(* CODESYS project tc3_vision.library
   TcLibraryId: Beckhoff Automation GmbH|Tc3_Vision|4.0.7.4
   Company: Beckhoff Automation GmbH
   DefaultNamespace: Tc3_Vision
   Version: 4.0.7.4
   Placeholder: Tc3_Vision
   Title: Tc3_Vision

Project tree, tasks and I/O mapping:
  Version/
    global variables Global_Version
  Function Blocks/
    Image Acquisition/
      function block FB_VN_GevCameraControl [ST]: ClearImageQueue, CloseCamera, FB_exit, FB_init, GetCalibPatternRef, GetCameraMatrix, GetCurrentImage, GetCurrentImageUndistorted, GetCurrentImageWithGvspInfo, GetCurrentImageWithGvspInfoUndistorted, GetCurrentImageWithTimestamps, GetDistortionCoefficients, GetLastImageFromQueue, GetOmittedImagesNum, GetRotationMatrix, GetState, GetTranslationVector, InitializeCamera, OpenCamera, Reset, ResetCameraFeatures, SetCameraMatrix, SetDistortionCoefficients, SetRotationMatrix, SetTranslationVector, StartAcquisition, StopAcquisition, TriggerImage
      function block FB_VN_FileSourceControl [ST]: FB_exit, FB_init, GetCurrentImage, GetCurrentImageAndFileName, StartAcquisition, StopAcquisition, Reset, GetState, TriggerImage, TriggerImageExp, TriggerImageByName
      function block FB_VN_SimpleCameraControl [ST]: FB_exit, FB_init, GetCurrentImage, GetState, Reset, StartAcquisition, StopAcquisition, TriggerImage
    File Access/
      function block FB_VN_InitializeFunction [ST]: FB_exit, FB_init
      function block FB_VN_ReadCalibrationPattern [ST]: FB_exit, FB_init
      function block FB_VN_ReadCalibrationResult [ST]: FB_exit, FB_init
      function block FB_VN_ReadContainer [ST]: FB_exit, FB_init
      function block FB_VN_ReadNeuralNetwork [ST]: FB_exit, FB_init
      function block FB_VN_ReadImage [ST]: FB_exit, FB_init
      function block FB_VN_ReadMlModel [ST]: FB_exit, FB_init
      function block FB_VN_WriteCalibrationResult [ST]: FB_exit, FB_init
      function block FB_VN_WriteContainer [ST]: FB_exit, FB_init
      function block FB_VN_WriteImage [ST]: FB_exit, FB_init
      function block FB_VN_WriteMlModel [ST]: FB_exit, FB_init
    Camera Register Access/
      function block FB_VN_ReadRegister_UDINT [ST]: FB_exit, FB_init
      function block FB_VN_WriteRegister_UDINT [ST]: FB_exit, FB_init
      function block FB_VN_ReadRegister_ULINT [ST]: FB_exit, FB_init
      function block FB_VN_WriteRegister_ULINT [ST]: FB_exit, FB_init
      function block FB_VN_ReadMemory [ST]: FB_exit, FB_init
      function block FB_VN_WriteMemory [ST]: FB_exit, FB_init
      function block FB_VN_ReadRegister_REAL [ST]: FB_exit, FB_init
      function block FB_VN_WriteRegister_REAL [ST]: FB_exit, FB_init
    Image Processing/
      function block FB_VN_GeneralizedHoughBallard [ST]: FB_exit, FB_init, Detect, SetCannyThreshold, SetInvAccuRatio, SetLevels, SetMinDist, SetTemplate, SetVotesThreshold
      function block FB_VN_SSIM [ST]: FB_exit, FB_init, Compute, SetReference
  Functions/
    Control Functions/
      function F_VN_StartAbsWatchdog [ST]
      function F_VN_StartAbsWatchdogExp [ST]
      function F_VN_StartRelWatchdog [ST]
      function F_VN_StartRelWatchdogExp [ST]
      function F_VN_StopWatchdog [ST]
    Image Segmentation/
      function F_VN_AdaptiveThreshold [ST]
      function F_VN_AdaptiveThresholdExp [ST]
      function F_VN_CheckColorRange [ST]
      function F_VN_DoubleThreshold [ST]
      function F_VN_SauvolaThreshold [ST]
      function F_VN_Threshold [ST]
      function F_VN_WatershedSegmentationExp [ST]
    Algebraic Container Operations/
      function F_VN_AddContainers [ST]
      F_VN_AddToContainerElements/
        function F_VN_AddToContainerElements_DINT [ST]
        function F_VN_AddToContainerElements_INT [ST]
        function F_VN_AddToContainerElements_LREAL [ST]
        function F_VN_AddToContainerElements_REAL [ST]
        function F_VN_AddToContainerElements_SINT [ST]
        function F_VN_AddToContainerElements_TcVnKeyPoint [ST]
        function F_VN_AddToContainerElements_TcVnPoint2_DINT [ST]
        function F_VN_AddToContainerElements_TcVnPoint2_LREAL [ST]
        function F_VN_AddToContainerElements_TcVnPoint2_REAL [ST]
        function F_VN_AddToContainerElements_TcVnPoint3_LREAL [ST]
        function F_VN_AddToContainerElements_TcVnPoint3_REAL [ST]
        function F_VN_AddToContainerElements_TcVnRectangle_DINT [ST]
        function F_VN_AddToContainerElements_TcVnRotatedRectangle [ST]
        function F_VN_AddToContainerElements_TcVnVector2_DINT [ST]
        function F_VN_AddToContainerElements_TcVnVector2_INT [ST]
        function F_VN_AddToContainerElements_TcVnVector2_REAL [ST]
        function F_VN_AddToContainerElements_TcVnVector2_SINT [ST]
        function F_VN_AddToContainerElements_TcVnVector2_UINT [ST]
        function F_VN_AddToContainerElements_TcVnVector2_USINT [ST]
        function F_VN_AddToContainerElements_TcVnVector3_INT [ST]
        function F_VN_AddToContainerElements_TcVnVector3_REAL [ST]
        function F_VN_AddToContainerElements_TcVnVector3_SINT [ST]
        function F_VN_AddToContainerElements_TcVnVector3_UINT [ST]
        function F_VN_AddToContainerElements_TcVnVector3_USINT [ST]
        function F_VN_AddToContainerElements_TcVnVector4_DINT [ST]
        function F_VN_AddToContainerElements_TcVnVector4_INT [ST]
        function F_VN_AddToContainerElements_TcVnVector4_LREAL [ST]
        function F_VN_AddToContainerElements_TcVnVector4_REAL [ST]
        function F_VN_AddToContainerElements_TcVnVector4_SINT [ST]
        function F_VN_AddToContainerElements_TcVnVector4_UINT [ST]
        function F_VN_AddToContainerElements_TcVnVector4_USINT [ST]
        function F_VN_AddToContainerElements_UDINT [ST]
        function F_VN_AddToContainerElements_UINT [ST]
        function F_VN_AddToContainerElements_ULINT [ST]
        function F_VN_AddToContainerElements_USINT [ST]
      function F_VN_BitwiseAndContainers [ST]
      function F_VN_BitwiseNotContainer [ST]
      function F_VN_BitwiseOrContainers [ST]
      function F_VN_BitwiseXorContainers [ST]
      function F_VN_DivideContainers [ST]
      function F_VN_DivideContainersExp [ST]
      function F_VN_MaxContainer [ST]
      function F_VN_MinContainer [ST]
      function F_VN_MultiplyContainers [ST]
      function F_VN_MultiplyWithContainerElements1 [ST]
      function F_VN_MultiplyWithContainerElements2 [ST]
      function F_VN_MultiplyWithContainerElements3 [ST]
      function F_VN_MultiplyWithContainerElements4 [ST]
      function F_VN_NegateContainer [ST]
      function F_VN_SubtractContainers [ST]
    Algebraic Image Operations/
      function F_VN_AddImages [ST]
      function F_VN_AddImagesWeighted [ST]
      function F_VN_AddImagesWeightedExp [ST]
      function F_VN_AddScalarToImage [ST]
      function F_VN_AddVectorToImage [ST]
      function F_VN_BitwiseAndImages [ST]
      function F_VN_BitwiseAndImagesExp [ST]
      function F_VN_BitwiseAndScalarWithImage [ST]
      function F_VN_BitwiseAndVectorWithImage [ST]
      function F_VN_BitwiseNotImage [ST]
      function F_VN_BitwiseNotImageExp [ST]
      function F_VN_BitwiseOrImages [ST]
      function F_VN_BitwiseOrImagesExp [ST]
      function F_VN_BitwiseOrScalarWithImage [ST]
      function F_VN_BitwiseOrVectorWithImage [ST]
      function F_VN_BitwiseXorImages [ST]
      function F_VN_BitwiseXorImagesExp [ST]
      function F_VN_BitwiseXorScalarWithImage [ST]
      function F_VN_BitwiseXorVectorWithImage [ST]
      function F_VN_BlendImages [ST]
      function F_VN_DivideImageByScalar [ST]
      function F_VN_DivideImageByVector [ST]
      function F_VN_DivideImages [ST]
      function F_VN_DivideScalarByImage [ST]
      function F_VN_DivideVectorByImage [ST]
      function F_VN_ElementwiseExp [ST]
      function F_VN_ElementwiseLog [ST]
      function F_VN_MaxImage [ST]
      function F_VN_MaxImageExp [ST]
      function F_VN_MaxImageWithScalar [ST]
      function F_VN_MaxImageWithScalarExp [ST]
      function F_VN_MaxImageWithVector [ST]
      function F_VN_MaxImageWithVectorExp [ST]
      function F_VN_MinImage [ST]
      function F_VN_MinImageExp [ST]
      function F_VN_MinImageWithScalar [ST]
      function F_VN_MinImageWithScalarExp [ST]
      function F_VN_MinImageWithVector [ST]
      function F_VN_MinImageWithVectorExp [ST]
      function F_VN_MultiplyImages [ST]
      function F_VN_MultiplyImageWithScalar [ST]
      function F_VN_MultiplyImageWithVector [ST]
      function F_VN_SubtractImageFromScalar [ST]
      function F_VN_SubtractImageFromVector [ST]
      function F_VN_SubtractImages [ST]
      function F_VN_SubtractScalarFromImage [ST]
      function F_VN_SubtractVectorFromImage [ST]
    Image Analysis/
      Object Detection/
        function F_VN_AdjustActiveContour [ST]
        function F_VN_DetectBlobs [ST]
        function F_VN_DetectBlobsExp [ST]
        function F_VN_FindContourHierarchyExp [ST]
        function F_VN_FindContours [ST]
        function F_VN_FindContoursExp [ST]
        function F_VN_HoughCircles [ST]
        function F_VN_HoughCirclesExp [ST]
        function F_VN_HoughLines [ST]
        function F_VN_HoughLinesExp [ST]
        function F_VN_HoughLinesP [ST]
        function F_VN_HoughLinesPExp [ST]
        function F_VN_MatchImageHuMoments [ST]
        function F_VN_MatchTemplate [ST]
        function F_VN_MatchTemplateExp [ST]
        function F_VN_MatchTemplateAndEvaluate [ST]
        function F_VN_MatchTemplateAndEvaluateExp [ST]
      function F_VN_CannyEdgeDetection [ST]
      function F_VN_CannyEdgeDetectionExp [ST]
      function F_VN_ConnectedComponents [ST]
      function F_VN_ConnectedComponentsExp [ST]
      function F_VN_ConnectedComponentsWithStats [ST]
      function F_VN_ConnectedComponentsWithStatsExp [ST]
      function F_VN_CountNonZeroPixels [ST]
      function F_VN_DistanceTransformation [ST]
      function F_VN_DistanceTransformationExp [ST]
      function F_VN_GetConnectedComponent [ST]
      function F_VN_GetConnectedComponentExp [ST]
      function F_VN_ImageAbsoluteAverage [ST]
      function F_VN_ImageAverage [ST]
      function F_VN_ImageAverageExp [ST]
      function F_VN_ImageAverageStdDev [ST]
      function F_VN_ImageAverageStdDevExp [ST]
      function F_VN_ImageCenterOfMass [ST]
      function F_VN_ImageCenterOfMassExp [ST]
      function F_VN_ImageMedian [ST]
      function F_VN_ImageMedianExp [ST]
      function F_VN_ImageMoments [ST]
      function F_VN_MaxPixelValue [ST]
      function F_VN_MaxPixelValueExp [ST]
      function F_VN_MinPixelValue [ST]
      function F_VN_MinPixelValueExp [ST]
      function F_VN_RegionOrientation [ST]
      function F_VN_RegionOrientationExp [ST]
      function F_VN_UprightInnerRectangle [ST]
      function F_VN_UprightInnerRectangleExp [ST]
    Measurement/
      function F_VN_AdjustSearchWindowOrientationToLinearEdge [ST]
      function F_VN_ClosestPointsBF [ST]
      function F_VN_LocateCircularArc [ST]
      function F_VN_LocateCircularArcExp [ST]
      function F_VN_LocateEdge [ST]
      function F_VN_LocateEdgeExp [ST]
      function F_VN_LocateEdges [ST]
      function F_VN_LocateEdgesExp [ST]
      function F_VN_LocateEllipse [ST]
      function F_VN_LocateEllipseExp [ST]
      function F_VN_MeasureAngleBetweenEdges [ST]
      function F_VN_MeasureAngleBetweenEdgesExp [ST]
      function F_VN_MeasureEdgeDistance [ST]
      function F_VN_MeasureEdgeDistanceExp [ST]
      function F_VN_MeasureMinEdgeDistance [ST]
      function F_VN_MeasureMinEdgeDistanceExp [ST]
    Basic Container Operations/
      function F_VN_AdvanceIterator [ST]
      F_VN_AppendToContainer/
        function F_VN_AppendToContainer_ITcVnContainer [ST]
        function F_VN_AppendToContainer_ITcVnForwardIterator [ST]
        function F_VN_AppendToContainer_DINT [ST]
        function F_VN_AppendToContainer_INT [ST]
        function F_VN_AppendToContainer_ITcVnImage [ST]
        function F_VN_AppendToContainer_LREAL [ST]
        function F_VN_AppendToContainer_REAL [ST]
        function F_VN_AppendToContainer_SINT [ST]
        function F_VN_AppendToContainer_TcVnDMatch [ST]
        function F_VN_AppendToContainer_TcVnKeyPoint [ST]
        function F_VN_AppendToContainer_TcVnPoint2_DINT [ST]
        function F_VN_AppendToContainer_TcVnPoint2_LREAL [ST]
        function F_VN_AppendToContainer_TcVnPoint2_REAL [ST]
        function F_VN_AppendToContainer_TcVnPoint3_LREAL [ST]
        function F_VN_AppendToContainer_TcVnPoint3_REAL [ST]
        function F_VN_AppendToContainer_TcVnRectangle_DINT [ST]
        function F_VN_AppendToContainer_TcVnRotatedRectangle [ST]
        function F_VN_AppendToContainer_TcVnVector2_DINT [ST]
        function F_VN_AppendToContainer_TcVnVector2_INT [ST]
        function F_VN_AppendToContainer_TcVnVector2_REAL [ST]
        function F_VN_AppendToContainer_TcVnVector2_SINT [ST]
        function F_VN_AppendToContainer_TcVnVector2_UINT [ST]
        function F_VN_AppendToContainer_TcVnVector2_USINT [ST]
        function F_VN_AppendToContainer_TcVnVector3_INT [ST]
        function F_VN_AppendToContainer_TcVnVector3_REAL [ST]
        function F_VN_AppendToContainer_TcVnVector3_SINT [ST]
        function F_VN_AppendToContainer_TcVnVector3_UINT [ST]
        function F_VN_AppendToContainer_TcVnVector3_USINT [ST]
        function F_VN_AppendToContainer_TcVnVector4_DINT [ST]
        function F_VN_AppendToContainer_TcVnVector4_INT [ST]
        function F_VN_AppendToContainer_TcVnVector4_LREAL [ST]
        function F_VN_AppendToContainer_TcVnVector4_REAL [ST]
        function F_VN_AppendToContainer_TcVnVector4_SINT [ST]
        function F_VN_AppendToContainer_TcVnVector4_UINT [ST]
        function F_VN_AppendToContainer_TcVnVector4_USINT [ST]
        function F_VN_AppendToContainer_UDINT [ST]
        function F_VN_AppendToContainer_UINT [ST]
        function F_VN_AppendToContainer_ULINT [ST]
        function F_VN_AppendToContainer_USINT [ST]
      function F_VN_CheckIfEmpty [ST]
      function F_VN_CheckIfIteratorIsAtEnd [ST]
      function F_VN_ConvertContainerType [ST]
      function F_VN_CopyContainer [ST]
      function F_VN_CopyContainerElementsConditional_ITcVnContainer [ST]
      function F_VN_CopyContainerElementsConditional_ITcVnForwardIterator [ST]
      function F_VN_CreateContainer [ST]
      function F_VN_CreateContainerFromArray [ST]
      function F_VN_EraseFromContainer [ST]
      function F_VN_ExportContainer [ST]
      function F_VN_ExportContainer_String [ST]
      function F_VN_ExportContainerSize [ST]
      function F_VN_ExportSubContainer [ST]
      function F_VN_ExportSubContainer_String [ST]
      function F_VN_ExportSubContainerSize [ST]
      function F_VN_ExtractContainerRange [ST]
      F_VN_FillContainer/
        function F_VN_FillContainer_DINT [ST]
        function F_VN_FillContainer_INT [ST]
        function F_VN_FillContainer_ITcVnImage [ST]
        function F_VN_FillContainer_LREAL [ST]
        function F_VN_FillContainer_REAL [ST]
        function F_VN_FillContainer_SINT [ST]
        function F_VN_FillContainer_TcVnDMatch [ST]
        function F_VN_FillContainer_TcVnKeyPoint [ST]
        function F_VN_FillContainer_TcVnPoint2_DINT [ST]
        function F_VN_FillContainer_TcVnPoint2_LREAL [ST]
        function F_VN_FillContainer_TcVnPoint2_REAL [ST]
        function F_VN_FillContainer_TcVnPoint3_LREAL [ST]
        function F_VN_FillContainer_TcVnPoint3_REAL [ST]
        function F_VN_FillContainer_TcVnRectangle_DINT [ST]
        function F_VN_FillContainer_TcVnRotatedRectangle [ST]
        function F_VN_FillContainer_TcVnVector2_DINT [ST]
        function F_VN_FillContainer_TcVnVector2_INT [ST]
        function F_VN_FillContainer_TcVnVector2_REAL [ST]
        function F_VN_FillContainer_TcVnVector2_SINT [ST]
        function F_VN_FillContainer_TcVnVector2_UINT [ST]
        function F_VN_FillContainer_TcVnVector2_USINT [ST]
        function F_VN_FillContainer_TcVnVector3_INT [ST]
        function F_VN_FillContainer_TcVnVector3_REAL [ST]
        function F_VN_FillContainer_TcVnVector3_SINT [ST]
        function F_VN_FillContainer_TcVnVector3_UINT [ST]
        function F_VN_FillContainer_TcVnVector3_USINT [ST]
        function F_VN_FillContainer_TcVnVector4_DINT [ST]
        function F_VN_FillContainer_TcVnVector4_INT [ST]
        function F_VN_FillContainer_TcVnVector4_LREAL [ST]
        function F_VN_FillContainer_TcVnVector4_REAL [ST]
        function F_VN_FillContainer_TcVnVector4_SINT [ST]
        function F_VN_FillContainer_TcVnVector4_UINT [ST]
        function F_VN_FillContainer_TcVnVector4_USINT [ST]
        function F_VN_FillContainer_UDINT [ST]
        function F_VN_FillContainer_UINT [ST]
        function F_VN_FillContainer_ULINT [ST]
        function F_VN_FillContainer_USINT [ST]
      F_VN_FillContainerExp/
        function F_VN_FillContainerExp_DINT [ST]
        function F_VN_FillContainerExp_INT [ST]
        function F_VN_FillContainerExp_ITcVnImage [ST]
        function F_VN_FillContainerExp_LREAL [ST]
        function F_VN_FillContainerExp_REAL [ST]
        function F_VN_FillContainerExp_SINT [ST]
        function F_VN_FillContainerExp_TcVnDMatch [ST]
        function F_VN_FillContainerExp_TcVnKeyPoint [ST]
        function F_VN_FillContainerExp_TcVnPoint2_DINT [ST]
        function F_VN_FillContainerExp_TcVnPoint2_LREAL [ST]
        function F_VN_FillContainerExp_TcVnPoint2_REAL [ST]
        function F_VN_FillContainerExp_TcVnPoint3_LREAL [ST]
        function F_VN_FillContainerExp_TcVnPoint3_REAL [ST]
        function F_VN_FillContainerExp_TcVnRectangle_DINT [ST]
        function F_VN_FillContainerExp_TcVnRotatedRectangle [ST]
        function F_VN_FillContainerExp_TcVnVector2_DINT [ST]
        function F_VN_FillContainerExp_TcVnVector2_INT [ST]
        function F_VN_FillContainerExp_TcVnVector2_REAL [ST]
        function F_VN_FillContainerExp_TcVnVector2_SINT [ST]
        function F_VN_FillContainerExp_TcVnVector2_UINT [ST]
        function F_VN_FillContainerExp_TcVnVector2_USINT [ST]
        function F_VN_FillContainerExp_TcVnVector3_INT [ST]
        function F_VN_FillContainerExp_TcVnVector3_REAL [ST]
        function F_VN_FillContainerExp_TcVnVector3_SINT [ST]
        function F_VN_FillContainerExp_TcVnVector3_UINT [ST]
        function F_VN_FillContainerExp_TcVnVector3_USINT [ST]
        function F_VN_FillContainerExp_TcVnVector4_DINT [ST]
        function F_VN_FillContainerExp_TcVnVector4_INT [ST]
        function F_VN_FillContainerExp_TcVnVector4_LREAL [ST]
        function F_VN_FillContainerExp_TcVnVector4_REAL [ST]
        function F_VN_FillContainerExp_TcVnVector4_SINT [ST]
        function F_VN_FillContainerExp_TcVnVector4_UINT [ST]
        function F_VN_FillContainerExp_TcVnVector4_USINT [ST]
        function F_VN_FillContainerExp_UDINT [ST]
        function F_VN_FillContainerExp_UINT [ST]
        function F_VN_FillContainerExp_ULINT [ST]
        function F_VN_FillContainerExp_USINT [ST]
      F_VN_GetAt/
        function F_VN_GetAt_ITcVnContainer [ST]
        function F_VN_GetAt_DINT [ST]
        function F_VN_GetAt_INT [ST]
        function F_VN_GetAt_ITcVnImage [ST]
        function F_VN_GetAt_LREAL [ST]
        function F_VN_GetAt_REAL [ST]
        function F_VN_GetAt_SINT [ST]
        function F_VN_GetAt_TcVnDMatch [ST]
        function F_VN_GetAt_TcVnKeyPoint [ST]
        function F_VN_GetAt_TcVnPoint2_DINT [ST]
        function F_VN_GetAt_TcVnPoint2_LREAL [ST]
        function F_VN_GetAt_TcVnPoint2_REAL [ST]
        function F_VN_GetAt_TcVnPoint3_LREAL [ST]
        function F_VN_GetAt_TcVnPoint3_REAL [ST]
        function F_VN_GetAt_TcVnRectangle_DINT [ST]
        function F_VN_GetAt_TcVnRotatedRectangle [ST]
        function F_VN_GetAt_TcVnVector2_DINT [ST]
        function F_VN_GetAt_TcVnVector2_INT [ST]
        function F_VN_GetAt_TcVnVector2_REAL [ST]
        function F_VN_GetAt_TcVnVector2_SINT [ST]
        function F_VN_GetAt_TcVnVector2_UINT [ST]
        function F_VN_GetAt_TcVnVector2_USINT [ST]
        function F_VN_GetAt_TcVnVector3_INT [ST]
        function F_VN_GetAt_TcVnVector3_REAL [ST]
        function F_VN_GetAt_TcVnVector3_SINT [ST]
        function F_VN_GetAt_TcVnVector3_UINT [ST]
        function F_VN_GetAt_TcVnVector3_USINT [ST]
        function F_VN_GetAt_TcVnVector4_DINT [ST]
        function F_VN_GetAt_TcVnVector4_INT [ST]
        function F_VN_GetAt_TcVnVector4_LREAL [ST]
        function F_VN_GetAt_TcVnVector4_REAL [ST]
        function F_VN_GetAt_TcVnVector4_SINT [ST]
        function F_VN_GetAt_TcVnVector4_UINT [ST]
        function F_VN_GetAt_TcVnVector4_USINT [ST]
        function F_VN_GetAt_UDINT [ST]
        function F_VN_GetAt_UINT [ST]
        function F_VN_GetAt_ULINT [ST]
        function F_VN_GetAt_USINT [ST]
      function F_VN_GetContainer [ST]
      function F_VN_GetContainerExp [ST]
      function F_VN_GetForwardIterator [ST]
      function F_VN_GetNumberOfElements [ST]
      function F_VN_GetRandomAccessIterator [ST]
      function F_VN_IncrementIterator [ST]
      F_VN_InsertIntoContainer/
        function F_VN_InsertIntoContainer_ITcVnContainer [ST]
        function F_VN_InsertIntoContainer_ITcVnForwardIterator [ST]
        function F_VN_InsertIntoContainer_DINT [ST]
        function F_VN_InsertIntoContainer_INT [ST]
        function F_VN_InsertIntoContainer_ITcVnImage [ST]
        function F_VN_InsertIntoContainer_LREAL [ST]
        function F_VN_InsertIntoContainer_REAL [ST]
        function F_VN_InsertIntoContainer_SINT [ST]
        function F_VN_InsertIntoContainer_TcVnDMatch [ST]
        function F_VN_InsertIntoContainer_TcVnKeyPoint [ST]
        function F_VN_InsertIntoContainer_TcVnPoint2_DINT [ST]
        function F_VN_InsertIntoContainer_TcVnPoint2_LREAL [ST]
        function F_VN_InsertIntoContainer_TcVnPoint2_REAL [ST]
        function F_VN_InsertIntoContainer_TcVnPoint3_LREAL [ST]
        function F_VN_InsertIntoContainer_TcVnPoint3_REAL [ST]
        function F_VN_InsertIntoContainer_TcVnRectangle_DINT [ST]
        function F_VN_InsertIntoContainer_TcVnRotatedRectangle [ST]
        function F_VN_InsertIntoContainer_TcVnVector2_DINT [ST]
        function F_VN_InsertIntoContainer_TcVnVector2_INT [ST]
        function F_VN_InsertIntoContainer_TcVnVector2_REAL [ST]
        function F_VN_InsertIntoContainer_TcVnVector2_SINT [ST]
        function F_VN_InsertIntoContainer_TcVnVector2_UINT [ST]
        function F_VN_InsertIntoContainer_TcVnVector2_USINT [ST]
        function F_VN_InsertIntoContainer_TcVnVector3_INT [ST]
        function F_VN_InsertIntoContainer_TcVnVector3_REAL [ST]
        function F_VN_InsertIntoContainer_TcVnVector3_SINT [ST]
        function F_VN_InsertIntoContainer_TcVnVector3_UINT [ST]
        function F_VN_InsertIntoContainer_TcVnVector3_USINT [ST]
        function F_VN_InsertIntoContainer_TcVnVector4_DINT [ST]
        function F_VN_InsertIntoContainer_TcVnVector4_INT [ST]
        function F_VN_InsertIntoContainer_TcVnVector4_LREAL [ST]
        function F_VN_InsertIntoContainer_TcVnVector4_REAL [ST]
        function F_VN_InsertIntoContainer_TcVnVector4_SINT [ST]
        function F_VN_InsertIntoContainer_TcVnVector4_UINT [ST]
        function F_VN_InsertIntoContainer_TcVnVector4_USINT [ST]
        function F_VN_InsertIntoContainer_UDINT [ST]
        function F_VN_InsertIntoContainer_UINT [ST]
        function F_VN_InsertIntoContainer_ULINT [ST]
        function F_VN_InsertIntoContainer_USINT [ST]
      function F_VN_IteratorDistance [ST]
      function F_VN_ReserveContainerMemory [ST]
      function F_VN_ReverseContainer [ST]
      F_VN_SetAt/
        function F_VN_SetAt_ITcVnContainer [ST]
        function F_VN_SetAt_DINT [ST]
        function F_VN_SetAt_INT [ST]
        function F_VN_SetAt_ITcVnImage [ST]
        function F_VN_SetAt_LREAL [ST]
        function F_VN_SetAt_REAL [ST]
        function F_VN_SetAt_SINT [ST]
        function F_VN_SetAt_TcVnDMatch [ST]
        function F_VN_SetAt_TcVnKeyPoint [ST]
        function F_VN_SetAt_TcVnPoint2_DINT [ST]
        function F_VN_SetAt_TcVnPoint2_LREAL [ST]
        function F_VN_SetAt_TcVnPoint2_REAL [ST]
        function F_VN_SetAt_TcVnPoint3_LREAL [ST]
        function F_VN_SetAt_TcVnPoint3_REAL [ST]
        function F_VN_SetAt_TcVnRectangle_DINT [ST]
        function F_VN_SetAt_TcVnRotatedRectangle [ST]
        function F_VN_SetAt_TcVnVector2_DINT [ST]
        function F_VN_SetAt_TcVnVector2_INT [ST]
        function F_VN_SetAt_TcVnVector2_REAL [ST]
        function F_VN_SetAt_TcVnVector2_SINT [ST]
        function F_VN_SetAt_TcVnVector2_UINT [ST]
        function F_VN_SetAt_TcVnVector2_USINT [ST]
        function F_VN_SetAt_TcVnVector3_INT [ST]
        function F_VN_SetAt_TcVnVector3_REAL [ST]
        function F_VN_SetAt_TcVnVector3_SINT [ST]
        function F_VN_SetAt_TcVnVector3_UINT [ST]
        function F_VN_SetAt_TcVnVector3_USINT [ST]
        function F_VN_SetAt_TcVnVector4_DINT [ST]
        function F_VN_SetAt_TcVnVector4_INT [ST]
        function F_VN_SetAt_TcVnVector4_LREAL [ST]
        function F_VN_SetAt_TcVnVector4_REAL [ST]
        function F_VN_SetAt_TcVnVector4_SINT [ST]
        function F_VN_SetAt_TcVnVector4_UINT [ST]
        function F_VN_SetAt_TcVnVector4_USINT [ST]
        function F_VN_SetAt_UDINT [ST]
        function F_VN_SetAt_UINT [ST]
        function F_VN_SetAt_ULINT [ST]
        function F_VN_SetAt_USINT [ST]
      function F_VN_SetContainer [ST]
      function F_VN_SetIteratorToBegin [ST]
    Geometric and Coordinate Transformations/
      function F_VN_AlignRotatedImageRegion [ST]
      function F_VN_AlignRotatedImageRegionExp [ST]
      function F_VN_ApplyRotationToAffineTransformation [ST]
      function F_VN_ApplyRotationToAffineTransformationExp [ST]
      function F_VN_ApplyScalingToAffineTransformation [ST]
      function F_VN_ApplyScalingToAffineTransformationExp [ST]
      function F_VN_ApplyTranslationToAffineTransformation [ST]
      function F_VN_ApplyTranslationToAffineTransformationExp [ST]
      function F_VN_ApplyYAxisInversionToAffineTransformation [ST]
      function F_VN_ApplyYAxisInversionToAffineTransformationExp [ST]
      Calibration/
        function F_VN_CalibrateCamera [ST]
        function F_VN_CalibrateCameraExp [ST]
        function F_VN_CalibrateCameraExp2 [ST]
        function F_VN_CalibrateCameraExp3 [ST]
        function F_VN_CalibrateCameraManually [ST]
        function F_VN_CalibrateCameraManuallyExp [ST]
        function F_VN_CalibrateCameraPlanar [ST]
        function F_VN_CalibrateCameraPlanarExp [ST]
        function F_VN_CalibrateLinescanCamera [ST]
        function F_VN_CalibrateLinescanCameraExp [ST]
        function F_VN_CompensateLensDistortion [ST]
        function F_VN_CompensateLensDistortionExp1 [ST]
        function F_VN_CompensateLensDistortionExp2 [ST]
        function F_VN_CompensateLensDistortionForPoints [ST]
        function F_VN_CompensateLensDistortionForPointsExp1 [ST]
        function F_VN_CompensateLensDistortionForPointsExp2 [ST]
        function F_VN_DetectPatternPoints [ST]
        function F_VN_DetectPatternPointsExp [ST]
        function F_VN_GenerateCalibrationPatternReferencePoints [ST]
        function F_VN_ImagePointsWorldDistance [ST]
        function F_VN_SolvePnP [ST]
        function F_VN_SolvePnPExp [ST]
        function F_VN_SortDetectedPatternPoints [ST]
        function F_VN_TransformCoordinatesPlanar_Container [ST]
        function F_VN_TransformCoordinatesPlanar_Point [ST]
        function F_VN_TransformCoordinatesImageToWorld_Container [ST]
        function F_VN_TransformCoordinatesImageToWorld_Point [ST]
        function F_VN_TransformCoordinatesWorldToImage_Container [ST]
        function F_VN_TransformCoordinatesWorldToImage_Point [ST]
      function F_VN_ConvertCartesianToPolarAngleImage [ST]
      function F_VN_ConvertCartesianToPolarAngleImageExp [ST]
      function F_VN_ConvertCartesianToPolarAngles [ST]
      function F_VN_ConvertCartesianToPolarAnglesExp [ST]
      function F_VN_ConvertCartesianToPolarImages [ST]
      function F_VN_ConvertCartesianToPolarImagesExp [ST]
      function F_VN_ConvertCartesianToPolarMagnitudeImage [ST]
      function F_VN_ConvertCartesianToPolarMagnitudes [ST]
      function F_VN_ConvertCartesianToPolarPoints [ST]
      function F_VN_ConvertCartesianToPolarPointsExp [ST]
      function F_VN_ConvertPolarToCartesianImages [ST]
      function F_VN_ConvertPolarToCartesianImagesExp [ST]
      function F_VN_ConvertPolarToCartesianPoints [ST]
      function F_VN_ConvertPolarToCartesianPointsExp [ST]
      function F_VN_DecomposeAffineTransformation [ST]
      function F_VN_DecomposeAffineTransformationExp [ST]
      function F_VN_DecomposeHomography [ST]
      function F_VN_DecomposeHomographyExp [ST]
      function F_VN_FlipImage [ST]
      function F_VN_GenerateAffineTransformationUnitMatrix2D [ST]
      function F_VN_GetAffineTransformation [ST]
      function F_VN_GetAffineTransformation2D [ST]
      function F_VN_GetAffineTransformation2DExp [ST]
      function F_VN_GetPerspectiveTransformation [ST]
      function F_VN_Homography [ST]
      function F_VN_HomographyExp [ST]
      function F_VN_InvertAffineTransformation [ST]
      function F_VN_PerspectiveTransformation [ST]
      function F_VN_PyramidDown [ST]
      function F_VN_PyramidUp [ST]
      function F_VN_RemapImageToLogPolarSpace [ST]
      function F_VN_RemapImageToLogPolarSpaceExp [ST]
      function F_VN_RemapImageToLogPolarSpaceExp2 [ST]
      function F_VN_RemapImageToPolarSpace [ST]
      function F_VN_RemapImageToPolarSpaceExp [ST]
      function F_VN_RemapImageToPolarSpaceExp2 [ST]
      function F_VN_ResizeImage [ST]
      function F_VN_ResizeImageExp [ST]
      function F_VN_RotateImage [ST]
      function F_VN_RotateImageExp [ST]
      function F_VN_RotateImageExp2 [ST]
      function F_VN_WarpAffine [ST]
      function F_VN_WarpAffineExp [ST]
      function F_VN_WarpAffine_Container [ST]
      function F_VN_WarpAffine_Point [ST]
      function F_VN_WarpAffine_Rectangle [ST]
      function F_VN_WarpPerspective [ST]
      function F_VN_WarpPerspective_Container [ST]
      function F_VN_WarpPerspectiveExp [ST]
      function F_VN_WarpPerspective_Point [ST]
      function F_VN_WarpPerspective_Rectangle [ST]
    Image Color and Contrast Processing/
      function F_VN_ApplyColorMap [ST]
      function F_VN_ApplyLut [ST]
      function F_VN_Clahe [ST]
      function F_VN_ClaheExp [ST]
      function F_VN_ConvertColorSpace [ST]
      function F_VN_GenerateColorMap [ST]
      function F_VN_GenerateCustomColorMap [ST]
      function F_VN_Histogram [ST]
      function F_VN_HistogramExp [ST]
      function F_VN_HistogramEqualization [ST]
      function F_VN_HistogramEqualizationExp [ST]
      function F_VN_InvertImageColor [ST]
      function F_VN_InvertImageColorExp [ST]
      function F_VN_NormalizeImage [ST]
      function F_VN_NormalizeImageExp [ST]
      function F_VN_NormalizeImageForDisplay [ST]
      function F_VN_ReferenceColorSimilarity_ITcVnColorModel [ST]
      function F_VN_ReferenceColorSimilarityExp_ITcVnColorModel [ST]
      function F_VN_ReferenceColorSimilarity_ITcVnMlModel [ST]
      function F_VN_ReferenceColorSimilarityExp_ITcVnMlModel [ST]
      function F_VN_ReferenceColorSimilarity_TcVnVector3_LREAL [ST]
      function F_VN_ReferenceColorSimilarityExp_TcVnVector3_LREAL [ST]
      function F_VN_TrainImageColor [ST]
      function F_VN_TrainImageColorExp [ST]
      function F_VN_TrainImageColorExp2 [ST]
      function F_VN_TrainImageColor_ITcVnMlModel [ST]
      function F_VN_TrainImageColorExp_ITcVnMlModel [ST]
      function F_VN_TrainImageColorExp2_ITcVnMlModel [ST]
      function F_VN_WhiteBalance [ST]
    Contour Analysis/
      function F_VN_ApproximatePolygon [ST]
      function F_VN_CheckIfPointIsInsideContour [ST]
      function F_VN_ContourArea [ST]
      function F_VN_ContourCenterOfMass [ST]
      function F_VN_ContourCircularity [ST]
      function F_VN_ContourCircularityExp [ST]
      function F_VN_ContourConvexity [ST]
      function F_VN_ContourEccentricity [ST]
      function F_VN_ContourElongation [ST]
      function F_VN_ContourExtremePoint [ST]
      function F_VN_ContourInertiaRatio [ST]
      function F_VN_ContourMoments [ST]
      function F_VN_ContourOrientation [ST]
      function F_VN_ContourOrientationExp [ST]
      function F_VN_ContourPerimeter [ST]
      function F_VN_ContourRoundness [ST]
      function F_VN_ConvexHullPoints [ST]
      function F_VN_ConvexHullPointsExp [ST]
      function F_VN_ConvexityDefects [ST]
      function F_VN_CustomElementWiseContainerOperation_ITcVnContainer [ST]
      function F_VN_CustomElementWiseContainerOperation_ITcVnForwardIterator [ST]
      function F_VN_EnclosingCircle [ST]
      function F_VN_EnclosingRectangle [ST]
      function F_VN_EnclosingTriangle [ST]
      function F_VN_FitEllipse [ST]
      function F_VN_FitLine [ST]
      function F_VN_FitLineExp [ST]
      function F_VN_FourierDescriptors [ST]
      function F_VN_MatchContours [ST]
      function F_VN_MatchContoursExp [ST]
      function F_VN_MatchContours1vsN [ST]
      function F_VN_MatchContours1vsNExp [ST]
      function F_VN_UprightBoundingRectangle [ST]
    Image Filtering/
      function F_VN_BilateralFilter [ST]
      function F_VN_BilateralFilterExp [ST]
      function F_VN_BoxFilter [ST]
      function F_VN_BoxFilterExp [ST]
      function F_VN_BrightBorderObjects [ST]
      function F_VN_CreateStructuringElement [ST]
      function F_VN_CustomFilter [ST]
      function F_VN_CustomFilterExp [ST]
      function F_VN_DarkBorderObjects [ST]
      function F_VN_FillHoles [ST]
      function F_VN_GaussianFilter [ST]
      function F_VN_GaussianFilterExp [ST]
      function F_VN_LaplacianFilter [ST]
      function F_VN_LaplacianFilterExp [ST]
      function F_VN_LocalMaxima [ST]
      function F_VN_LocalMinima [ST]
      function F_VN_MedianFilter [ST]
      function F_VN_MorphologicalOperator [ST]
      function F_VN_RemoveLocalMaxima [ST]
      function F_VN_RemoveLocalMinima [ST]
      function F_VN_ScharrFilter [ST]
      function F_VN_ScharrFilterExp [ST]
      function F_VN_SeparableCustomFilter [ST]
      function F_VN_SeparableCustomFilterExp [ST]
      function F_VN_SobelFilter [ST]
      function F_VN_SobelFilterExp [ST]
      function F_VN_VarianceFilter [ST]
      function F_VN_VarianceFilterExp [ST]
    Miscellaneous/
      function F_VN_CheckFunctionInitialization [ST]
      function F_VN_ClipLineToBoundary [ST]
      function F_VN_ClipLineToBoundary_ITcVnImage [ST]
      function F_VN_ClipLineToBoundary_TcVnRectangle_DINT [ST]
      function F_VN_ConvertITcUnknownToITcVnBitmapExport [ST]
      function F_VN_ConvertITcUnknownToITcVnContainer [ST]
      function F_VN_ConvertITcUnknownToITcVnImage [ST]
      function F_VN_ConvertITcUnknownToITcVnMlModel [ST]
      function F_VN_DeinitializeFunction [ST]
      function F_VN_GetTimestamp [ST]
      function F_VN_HuMomentInvariants [ST]
      function F_VN_InitMatrixStruct [ST]
      function F_VN_InvertMatrix3x3 [ST]
      function F_VN_LineIntersectionPoint [ST]
      function F_VN_LineIntersectionPointAndAngle [ST]
      function F_VN_MultiplyMatrices [ST]
      function F_VN_OrthogonalVector_TcVnVector2_DINT [ST]
      function F_VN_OrthogonalVector_TcVnVector2_LREAL [ST]
      function F_VN_OrthogonalVector_TcVnVector2_REAL [ST]
      function F_VN_PointToLineDistance_TcVnPoint2_DINT [ST]
      function F_VN_PointToLineDistance_TcVnPoint2_LREAL [ST]
      function F_VN_PointToLineDistance_TcVnPoint2_REAL [ST]
      function F_VN_PointToPointDirection_TcVnPoint2_DINT [ST]
      function F_VN_PointToPointDirection_TcVnPoint2_LREAL [ST]
      function F_VN_PointToPointDirection_TcVnPoint2_REAL [ST]
      function F_VN_PointToPointDistance_TcVnPoint2_DINT [ST]
      function F_VN_PointToPointDistance_TcVnPoint2_LREAL [ST]
      function F_VN_PointToPointDistance_TcVnPoint2_REAL [ST]
      function F_VN_RotatedRectangleCorners [ST]
      function F_VN_RotatedRectangleIntersection [ST]
      function F_VN_SetRngSeed [ST]
      function F_VN_UpdateTimestamp [ST]
    Basic Image Operations/
      function F_VN_CombineImageChannels [ST]
      function F_VN_ConvertElementType [ST]
      function F_VN_ConvertElementTypeExp [ST]
      function F_VN_CopyImage [ST]
      function F_VN_CopyImageRegion [ST]
      function F_VN_CopyImageRegionToRegion [ST]
      function F_VN_CopyIntoDisplayableImage [ST]
      function F_VN_CreateAssociatedImage [ST]
      function F_VN_CreateEmptyImage [ST]
      function F_VN_CreateImage [ST]
      function F_VN_CreateNDimensionalImage [ST]
      function F_VN_CreateImageAndSetPixels [ST]
      function F_VN_CreateNDimensionalImageAndSetPixels [ST]
      function F_VN_CreateImageFromArray [ST]
      function F_VN_CreateNDimensionalImageFromArray [ST]
      function F_VN_ExportImage [ST]
      function F_VN_ExportImageSize [ST]
      function F_VN_ExportImageAsBmp [ST]
      function F_VN_ExportImageAsBmpExp [ST]
      function F_VN_ExportImageAsBmpSize [ST]
      function F_VN_ExportImageAsBmpSizeExp [ST]
      function F_VN_FuseImages [ST]
      function F_VN_FuseImagesArray [ST]
      function F_VN_GetImageChannel [ST]
      function F_VN_GetImageHeight [ST]
      function F_VN_GetImageInfo [ST]
      function F_VN_GetImageWidth [ST]
      function F_VN_GetLayoutInfo [ST]
      function F_VN_GetPixel [ST]
      function F_VN_GetPixelFormat [ST]
      function F_VN_GetRoi [ST]
      function F_VN_MixImageChannels [ST]
      function F_VN_PadImageBorder [ST]
      function F_VN_PadImageBorderExp [ST]
      function F_VN_ReinterpretUnsupportedImage [ST]
      function F_VN_ResetRoi [ST]
      function F_VN_SetImageChannel [ST]
      function F_VN_SetPixel [ST]
      function F_VN_SetPixels [ST]
      function F_VN_SetPixelsExp [ST]
      function F_VN_SetRoi [ST]
      function F_VN_SetRoi_TcVnRectangle_DINT [ST]
      function F_VN_SetRoi_TcVnRectangle_UDINT [ST]
      function F_VN_SplitImageChannels [ST]
      function F_VN_TransformIntoDisplayableImage [ST]
      function F_VN_TransformIntoDisplayableImageExp [ST]
    Container Statistics/
      function F_VN_ContainerAverage [ST]
      function F_VN_ContainerAverageElementwise2 [ST]
      function F_VN_ContainerAverageElementwise3 [ST]
      function F_VN_ContainerAverageElementwise4 [ST]
      function F_VN_ContainerAverageVariance [ST]
      function F_VN_ContainerAverageVarianceElementwise2 [ST]
      function F_VN_ContainerAverageVarianceElementwise3 [ST]
      function F_VN_ContainerAverageVarianceElementwise4 [ST]
      function F_VN_MaxElement [ST]
      F_VN_MaxElementElementwise/
        function F_VN_MaxElementElementwise_DINT [ST]
        function F_VN_MaxElementElementwise_INT [ST]
        function F_VN_MaxElementElementwise_LREAL [ST]
        function F_VN_MaxElementElementwise_REAL [ST]
        function F_VN_MaxElementElementwise_SINT [ST]
        function F_VN_MaxElementElementwise_TcVnPoint2_DINT [ST]
        function F_VN_MaxElementElementwise_TcVnPoint2_LREAL [ST]
        function F_VN_MaxElementElementwise_TcVnPoint2_REAL [ST]
        function F_VN_MaxElementElementwise_TcVnPoint3_LREAL [ST]
        function F_VN_MaxElementElementwise_TcVnPoint3_REAL [ST]
        function F_VN_MaxElementElementwise_TcVnVector2_DINT [ST]
        function F_VN_MaxElementElementwise_TcVnVector2_INT [ST]
        function F_VN_MaxElementElementwise_TcVnVector2_REAL [ST]
        function F_VN_MaxElementElementwise_TcVnVector2_SINT [ST]
        function F_VN_MaxElementElementwise_TcVnVector2_UINT [ST]
        function F_VN_MaxElementElementwise_TcVnVector2_USINT [ST]
        function F_VN_MaxElementElementwise_TcVnVector3_INT [ST]
        function F_VN_MaxElementElementwise_TcVnVector3_REAL [ST]
        function F_VN_MaxElementElementwise_TcVnVector3_SINT [ST]
        function F_VN_MaxElementElementwise_TcVnVector3_UINT [ST]
        function F_VN_MaxElementElementwise_TcVnVector3_USINT [ST]
        function F_VN_MaxElementElementwise_TcVnVector4_DINT [ST]
        function F_VN_MaxElementElementwise_TcVnVector4_INT [ST]
        function F_VN_MaxElementElementwise_TcVnVector4_LREAL [ST]
        function F_VN_MaxElementElementwise_TcVnVector4_REAL [ST]
        function F_VN_MaxElementElementwise_TcVnVector4_SINT [ST]
        function F_VN_MaxElementElementwise_TcVnVector4_UINT [ST]
        function F_VN_MaxElementElementwise_TcVnVector4_USINT [ST]
        function F_VN_MaxElementElementwise_UDINT [ST]
        function F_VN_MaxElementElementwise_UINT [ST]
        function F_VN_MaxElementElementwise_ULINT [ST]
        function F_VN_MaxElementElementwise_USINT [ST]
      function F_VN_MedianElement [ST]
      F_VN_MedianElementElementwise/
        function F_VN_MedianElementElementwise_DINT [ST]
        function F_VN_MedianElementElementwise_INT [ST]
        function F_VN_MedianElementElementwise_LREAL [ST]
        function F_VN_MedianElementElementwise_REAL [ST]
        function F_VN_MedianElementElementwise_SINT [ST]
        function F_VN_MedianElementElementwise_TcVnPoint2_DINT [ST]
        function F_VN_MedianElementElementwise_TcVnPoint2_LREAL [ST]
        function F_VN_MedianElementElementwise_TcVnPoint2_REAL [ST]
        function F_VN_MedianElementElementwise_TcVnPoint3_LREAL [ST]
        function F_VN_MedianElementElementwise_TcVnPoint3_REAL [ST]
        function F_VN_MedianElementElementwise_TcVnVector2_DINT [ST]
        function F_VN_MedianElementElementwise_TcVnVector2_INT [ST]
        function F_VN_MedianElementElementwise_TcVnVector2_REAL [ST]
        function F_VN_MedianElementElementwise_TcVnVector2_SINT [ST]
        function F_VN_MedianElementElementwise_TcVnVector2_UINT [ST]
        function F_VN_MedianElementElementwise_TcVnVector2_USINT [ST]
        function F_VN_MedianElementElementwise_TcVnVector3_INT [ST]
        function F_VN_MedianElementElementwise_TcVnVector3_REAL [ST]
        function F_VN_MedianElementElementwise_TcVnVector3_SINT [ST]
        function F_VN_MedianElementElementwise_TcVnVector3_UINT [ST]
        function F_VN_MedianElementElementwise_TcVnVector3_USINT [ST]
        function F_VN_MedianElementElementwise_TcVnVector4_DINT [ST]
        function F_VN_MedianElementElementwise_TcVnVector4_INT [ST]
        function F_VN_MedianElementElementwise_TcVnVector4_LREAL [ST]
        function F_VN_MedianElementElementwise_TcVnVector4_REAL [ST]
        function F_VN_MedianElementElementwise_TcVnVector4_SINT [ST]
        function F_VN_MedianElementElementwise_TcVnVector4_UINT [ST]
        function F_VN_MedianElementElementwise_TcVnVector4_USINT [ST]
        function F_VN_MedianElementElementwise_UDINT [ST]
        function F_VN_MedianElementElementwise_UINT [ST]
        function F_VN_MedianElementElementwise_ULINT [ST]
        function F_VN_MedianElementElementwise_USINT [ST]
      function F_VN_MinElement [ST]
      F_VN_MinElementElementwise/
        function F_VN_MinElementElementwise_DINT [ST]
        function F_VN_MinElementElementwise_INT [ST]
        function F_VN_MinElementElementwise_LREAL [ST]
        function F_VN_MinElementElementwise_REAL [ST]
        function F_VN_MinElementElementwise_SINT [ST]
        function F_VN_MinElementElementwise_TcVnPoint2_DINT [ST]
        function F_VN_MinElementElementwise_TcVnPoint2_LREAL [ST]
        function F_VN_MinElementElementwise_TcVnPoint2_REAL [ST]
        function F_VN_MinElementElementwise_TcVnPoint3_LREAL [ST]
        function F_VN_MinElementElementwise_TcVnPoint3_REAL [ST]
        function F_VN_MinElementElementwise_TcVnVector2_DINT [ST]
        function F_VN_MinElementElementwise_TcVnVector2_INT [ST]
        function F_VN_MinElementElementwise_TcVnVector2_REAL [ST]
        function F_VN_MinElementElementwise_TcVnVector2_SINT [ST]
        function F_VN_MinElementElementwise_TcVnVector2_UINT [ST]
        function F_VN_MinElementElementwise_TcVnVector2_USINT [ST]
        function F_VN_MinElementElementwise_TcVnVector3_INT [ST]
        function F_VN_MinElementElementwise_TcVnVector3_REAL [ST]
        function F_VN_MinElementElementwise_TcVnVector3_SINT [ST]
        function F_VN_MinElementElementwise_TcVnVector3_UINT [ST]
        function F_VN_MinElementElementwise_TcVnVector3_USINT [ST]
        function F_VN_MinElementElementwise_TcVnVector4_DINT [ST]
        function F_VN_MinElementElementwise_TcVnVector4_INT [ST]
        function F_VN_MinElementElementwise_TcVnVector4_LREAL [ST]
        function F_VN_MinElementElementwise_TcVnVector4_REAL [ST]
        function F_VN_MinElementElementwise_TcVnVector4_SINT [ST]
        function F_VN_MinElementElementwise_TcVnVector4_UINT [ST]
        function F_VN_MinElementElementwise_TcVnVector4_USINT [ST]
        function F_VN_MinElementElementwise_UDINT [ST]
        function F_VN_MinElementElementwise_UINT [ST]
        function F_VN_MinElementElementwise_ULINT [ST]
        function F_VN_MinElementElementwise_USINT [ST]
    Fourier Analysis/
      function F_VN_CreateBandpassButterworthFilter [ST]
      function F_VN_CreateBandpassGaussianFilter [ST]
      function F_VN_CreateBandrejectButterworthFilter [ST]
      function F_VN_CreateBandrejectGaussianFilter [ST]
      function F_VN_CreateHighpassButterworthFilter [ST]
      function F_VN_CreateHighpassGaussianFilter [ST]
      function F_VN_CreateLowpassButterworthFilter [ST]
      function F_VN_CreateLowpassGaussianFilter [ST]
      function F_VN_Dft [ST]
      function F_VN_InverseDft [ST]
      function F_VN_OptimalDftSize [ST]
    Machine Learning/
      function F_VN_CreateBoostClassifier [ST]
      function F_VN_CreateBoostClassifierExp [ST]
      function F_VN_CreateBoostClassifierExp2 [ST]
      function F_VN_CreateKmppModel [ST]
      function F_VN_CreateKmppModelExp [ST]
      function F_VN_CreateKnnModel [ST]
      function F_VN_CreateLbgModel [ST]
      function F_VN_CreateLbgModelExp [ST]
      function F_VN_CreateLdaTransform [ST]
      function F_VN_CreateLdaTransformViaComponentNum [ST]
      function F_VN_CreateNbcModel [ST]
      function F_VN_CreatePcaTransform [ST]
      function F_VN_CreatePcaTransformViaComponentNum [ST]
      function F_VN_CreatePcaTransformViaVariance [ST]
      function F_VN_CreateRTreesModel [ST]
      function F_VN_CreateRTreesModelExp [ST]
      function F_VN_CreateRTreesModelExp2 [ST]
      function F_VN_CreateStaModel [ST]
      function F_VN_CreateStaModelExp [ST]
      function F_VN_CreateStaModelExp2 [ST]
      function F_VN_CreateSvmModel [ST]
      function F_VN_CreateSvmModelExp [ST]
      function F_VN_CreateSvmModelExp2 [ST]
      function F_VN_CreateSvmSgdClassifier [ST]
      function F_VN_CreateSvmSgdClassifierExp [ST]
      function F_VN_FeatureTransform [ST]
      function F_VN_GetBatchClusters [ST]
      function F_VN_GetBatchClustersExp [ST]
      function F_VN_GetBatchNovelties [ST]
      function F_VN_GetClusterCenter [ST]
      function F_VN_GetClusterNum [ST]
      function F_VN_GetFeatureScales [ST]
      function F_VN_GetSampleCluster [ST]
      function F_VN_GetSampleClusterExp [ST]
      function F_VN_GetSampleNovelty [ST]
      function F_VN_InverseFeatureScaling [ST]
      function F_VN_InverseFeatureScaling_REAL [ST]
      function F_VN_InverseFeatureScalingExp [ST]
      function F_VN_InverseFeatureScalingExp_REAL [ST]
      function F_VN_InverseFeatureTransform [ST]
      function F_VN_PredictBatch [ST]
      function F_VN_PredictBatchExp [ST]
      function F_VN_PredictSampleClass [ST]
      function F_VN_PredictSampleClassExp [ST]
      function F_VN_PredictSampleScalar [ST]
      function F_VN_PredictSampleScalarExp [ST]
      function F_VN_PredictSampleVector [ST]
      function F_VN_PredictSampleVectorExp [ST]
      function F_VN_FeatureScaling [ST]
      function F_VN_FeatureScalingExp [ST]
      function F_VN_TrainBatch [ST]
      function F_VN_TrainBatchClusters [ST]
      function F_VN_TrainSample [ST]
      function F_VN_TrainSampleClass [ST]
      function F_VN_TrainSampleCluster [ST]
      function F_VN_TrainSampleScalar [ST]
      function F_VN_TrainSampleVector [ST]
    Drawing/
      function F_VN_DrawArrow [ST]
      function F_VN_DrawArrow_TcVnVector4_DINT [ST]
      function F_VN_DrawArrowExp [ST]
      function F_VN_DrawArrowExp_TcVnVector4_DINT [ST]
      function F_VN_DrawCircle [ST]
      function F_VN_DrawCircleExp [ST]
      function F_VN_DrawCircles [ST]
      function F_VN_DrawCirclesExp [ST]
      function F_VN_DrawCircularArc [ST]
      function F_VN_DrawCircularArcExp [ST]
      function F_VN_DrawComponents [ST]
      function F_VN_DrawComponentsExp [ST]
      function F_VN_DrawContours [ST]
      function F_VN_DrawContoursExp [ST]
      function F_VN_DrawEllipse [ST]
      function F_VN_DrawEllipseExp [ST]
      function F_VN_DrawKeypoints [ST]
      function F_VN_DrawKeypointsExp [ST]
      function F_VN_DrawLine [ST]
      function F_VN_DrawLineExp [ST]
      function F_VN_DrawLine_TcVnVector4_DINT [ST]
      function F_VN_DrawLineExp_TcVnVector4_DINT [ST]
      function F_VN_DrawLine_TcVnVector4_LREAL [ST]
      function F_VN_DrawLineExp_TcVnVector4_LREAL [ST]
      function F_VN_DrawLines [ST]
      function F_VN_DrawLinesExp [ST]
      function F_VN_DrawMatches [ST]
      function F_VN_DrawMatchesExp [ST]
      function F_VN_DrawOrientation [ST]
      function F_VN_DrawOrientationExp [ST]
      function F_VN_DrawPoint [ST]
      function F_VN_DrawPointExp [ST]
      function F_VN_DrawPoints [ST]
      function F_VN_DrawPointsExp [ST]
      function F_VN_DrawPolygon [ST]
      function F_VN_DrawPolygonExp [ST]
      function F_VN_DrawRectangle [ST]
      function F_VN_DrawRectangle_TcVnRectangle_DINT [ST]
      function F_VN_DrawRectangle_TcVnRectangle_UDINT [ST]
      function F_VN_DrawRotatedRectangle [ST]
      function F_VN_DrawRotatedRectangleExp [ST]
      function F_VN_FillCircle [ST]
      function F_VN_FillContours [ST]
      function F_VN_FillEllipse [ST]
      function F_VN_FillPolygon [ST]
      function F_VN_FillRectangle [ST]
      function F_VN_FillRotatedRectangle [ST]
      function F_VN_PlotIntensityProfile [ST]
      function F_VN_PlotIntensityProfileExp [ST]
      function F_VN_PutLabel [ST]
      function F_VN_PutLabelExp [ST]
      function F_VN_PutText [ST]
      function F_VN_PutTextExp [ST]
    Neural Network/
      function F_VN_ConvertDataLayout [ST]
      function F_VN_ReshapeImage [ST]
      function F_VN_Sigmoid [ST]
      function F_VN_SigmoidExp [ST]
      function F_VN_SoftMax [ST]
      function F_VN_NonMaxSuppression [ST]
      function F_VN_NonMaxSuppressionExp [ST]
      function F_VN_ExecuteNeuralNetwork [ST]
      function F_VN_ExecuteNeuralNetwork_MI [ST]
      function F_VN_ExecuteNeuralNetwork_MultiLayerOutput [ST]
      function F_VN_ExecuteNeuralNetwork_MO [ST]
      function F_VN_ExecuteNeuralNetwork_MIMO_String [ST]
      function F_VN_ExecuteNeuralNetwork_SingleLayerOutput [ST]
      function F_VN_ExecuteNeuralNetwork_SO [ST]
      function F_VN_ExecuteNeuralNetwork_MISO [ST]
      function F_VN_GetNeuralNetworkLayerNames [ST]
      function F_VN_GetNeuralNetworkLayerNamesExp [ST]
      function F_VN_GetNeuralNetworkLayerNamesExp_String [ST]
      function F_VN_Reduce [ST]
      function F_VN_ReduceArg [ST]
    Keypoint Features/
      function F_VN_FilterGoodMatches [ST]
      function F_VN_FindReferenceKeyPointsInImage [ST]
      function F_VN_FindReferenceKeyPointsInImageExp [ST]
      function F_VN_FindReferenceKeyPointsInImageAKAZE [ST]
      function F_VN_FindReferenceKeyPointsInImageAKAZEExp [ST]
      function F_VN_FindReferenceKeyPointsInImageBRISK [ST]
      function F_VN_FindReferenceKeyPointsInImageBRISKExp [ST]
      function F_VN_FindReferenceKeyPointsInImageORB [ST]
      function F_VN_FindReferenceKeyPointsInImageORBExp [ST]
      function F_VN_GetMatchCoordinates [ST]
      function F_VN_KeyPointsAGAST [ST]
      function F_VN_KeyPointsAGASTExp [ST]
      function F_VN_KeyPointsAndDescriptorsAKAZE [ST]
      function F_VN_KeyPointsAndDescriptorsAKAZEExp [ST]
      function F_VN_KeyPointsAndDescriptorsBRISK [ST]
      function F_VN_KeyPointsAndDescriptorsBRISKExp [ST]
      function F_VN_KeyPointsAndDescriptorsKAZE [ST]
      function F_VN_KeyPointsAndDescriptorsKAZEExp [ST]
      function F_VN_KeyPointsAndDescriptorsORB [ST]
      function F_VN_KeyPointsAndDescriptorsORBExp [ST]
      function F_VN_KeyPointsFAST [ST]
      function F_VN_KeyPointsFASTExp [ST]
      function F_VN_KeyPointsGFTT [ST]
      function F_VN_KeyPointsGFTTExp [ST]
      function F_VN_KeyPointsMSER [ST]
      function F_VN_KeyPointsMSERExp [ST]
      function F_VN_KeyPointsSB [ST]
      function F_VN_KeyPointsSBExp [ST]
      function F_VN_MatchDescriptorsBF [ST]
      function F_VN_MatchDescriptorsBFExp [ST]
      function F_VN_MatchDescriptorsFlannLsh [ST]
      function F_VN_MatchDescriptorsFlannLshExp [ST]
      function F_VN_MatchDescriptorsKnnBF [ST]
      function F_VN_MatchDescriptorsKnnBFExp [ST]
      function F_VN_MatchDescriptorsKnnFlannLsh [ST]
      function F_VN_MatchDescriptorsKnnFlannLshExp [ST]
      function F_VN_RegionsMSER [ST]
      function F_VN_RegionsMSERExp [ST]
    Code Quality/
      function F_VN_GradeBarcode [ST]
      function F_VN_GradeBarcodeExp [ST]
      function F_VN_GradeDataMatrixCode [ST]
      function F_VN_GradeDataMatrixCodeExp [ST]
      function F_VN_GradeQRCode [ST]
      function F_VN_GradeQRCodeExp [ST]
    Texture Analysis/
      function F_VN_Granulometry [ST]
      function F_VN_HaralickFeatures [ST]
    OCR/
      function F_VN_OCR [ST]
      function F_VN_OCRExp [ST]
    Code Reading/
      function F_VN_ReadBarcode [ST]
      function F_VN_ReadBarcodeExp [ST]
      function F_VN_ReadBarcodeExp2 [ST]
      function F_VN_ReadDataMatrixCode [ST]
      function F_VN_ReadDataMatrixCodeExp [ST]
      function F_VN_ReadDataMatrixCodeExp2 [ST]
      function F_VN_ReadDataMatrixCodeRoi [ST]
      function F_VN_ReadDataMatrixCodeRoiExp [ST]
      function F_VN_ReadPharmaCode [ST]
      function F_VN_ReadPharmaCodeExp [ST]
      function F_VN_ReadPharmaCodeExp2 [ST]
      function F_VN_ReadQRCode [ST]
      function F_VN_ReadQRCodeExp [ST]
      function F_VN_ReadQRCodeExp2 [ST]
  Data Types/
    Enumerations/
      data type ETcVn2dCodeSearchStrategy
      data type ETcVnAdaptiveThresholdMethod
      data type ETcVnBarcodeSearchDirection
      data type ETcVnBarcodeType
      data type ETcVnBlobCombination
      data type ETcVnBoostClassifierType
      data type ETcVnBorderInterpolationMethod
      data type ETcVnCalibrationPattern
      data type ETcVnCalibrationPatternOrigin
      data type ETcVnCameraState
      data type ETcVnClusteringAlgorithm
      data type ETcVnColorMap
      data type ETcVnColorMapSize
      data type ETcVnColorSpaceTransform
      data type ETcVnColorTrainingMethod
      data type ETcVnConnectedComponentsAlgorithm
      data type ETcVnContainerExportFormat
      data type ETcVnContourApproximationMethod
      data type ETcVnCircularityCalculationMethod
      data type ETcVnContoursMatchComparisonMethod
      data type ETcVnContourRetrievalMode
      data type ETcVnDataLayout
      data type ETcVnLayerNameType
      data type ETcVnDataMatrixOptions
      data type ETcVnDiffusivityTypeKAZE
      data type ETcVnDistanceTransformationLabel
      data type ETcVnDistanceTransformationMask
      data type ETcVnDistanceType
      data type ETcVnDrawShape
      data type ETcVnDrawMatchesFlags
      data type ETcVnEdgeDetectionAlgorithm
      data type ETcVnEdgeDirection
      data type ETcVnEstimationAlgorithm
      data type ETcVnExtremePointDirection
      data type ETcVnFeatureDescriptorTypeAKAZE
      data type ETcVnFeatureScoreTypeORB
      data type ETcVnFlipAxis
      data type ETcVnFilterDirection
      data type ETcVnFontType
      data type ETcVnHoughMethod
      data type ETcVnInitializableFunction
      data type ETcVnInterpolationType
      data type ETcVnKnn
      data type ETcVnLineType
      data type ETcVnMorphologicalOperator
      data type ETcVnNbc
      data type ETcVnNormalizationType
      data type ETcVnFeatureScalingType
      data type ETcVnOcrModelType
      data type ETcVnOcrOptions
      data type ETcVnOrientationMethod
      data type ETcVnPaddingMode
      data type ETcVnPixelConnectivity
      data type ETcVnPrototypeClusterer
      data type ETcVnRectangleIntersection
      data type ETcVnReduceType
      data type ETcVnRotationAngle
      data type ETcVnRTrees
      data type ETcVnSignedNormalization
      data type ETcVnSolvePnPMethod
      data type ETcVnSta
      data type ETcVnStructuringElementShape
      data type ETcVnSvm
      data type ETcVnSvmKernelType
      data type ETcVnSvmSgdClassifierType
      data type ETcVnSvmSgdClassifierMarginType
      data type ETcVnTemplateMatchMethod
      data type ETcVnThresholdType
      data type ETcVnTimestamp
      data type ETcVnVectorCompareMethod
      data type ETcVnKeypointDetectionTypeAGAST
      data type ETcVnKeypointDetectionTypeFAST
      data type ETcVnWorldCoordinateSystem
    Structs/
      data type TcVnCodeGrades1D
      data type TcVnCodeGradesDM
      data type TcVnCodeGradesQR
      data type TcVnParamsAGAST
      data type TcVnParamsAKAZE
      data type TcVnParamsBlobDetection
      data type TcVnParamsBRISK
      data type TcVnParamsFAST
      data type TcVnParamsGFTT
      data type TcVnParamsKAZE
      data type TcVnParamsMSER
      data type TcVnParamsORB
      data type TcVnParamsSB
  Interfaces/
    Containers/
      Function Blocks/
        interface ITcVnCustomContainerOperation_ITcVnContainer: Execute
        interface ITcVnCustomContainerOperation_ITcVnForwardIterator: Execute
        interface ITcVnCustomElementCondition_ITcVnContainer: Condition
        interface ITcVnCustomElementCondition_ITcVnForwardIterator: Condition
    Machine Learning/
      interface ITcVnColorModel: TrainImageColor, ClassifyImageColor
  Global Variables/
    global variables Global_Variables
    global variables TC3_VISION_IID_LIST
*)

// Data Types/Enumerations/ETcVn2dCodeSearchStrategy

(* Offers search strategies for 2d code reading (multiple TCVN_CSS_XXX_INVERTED or multiple TCVN_CSS_XXX_FLIPPED cannot be combined). *)
	{attribute 'TcIecLibraryType'}
{attribute 'Namespace' := 'Tc3_Vision'}
TYPE ETcVn2dCodeSearchStrategy : (
	TCVN_CSS_DEFAULT:=1, 	(* The algorithm searches for codes using the default searching strategy, all other flags are ignored (dependant on code type). *)
	TCVN_CSS_ONLY_NOT_INVERTED:=8, 	(* The algorithm searches for codes only in the non-inverted image. *)
	TCVN_CSS_FIRST_NOT_INVERTED:=10, 	(* The algorithm first searches for codes in the non-inverted and then in the inverted image. *)
	TCVN_CSS_ONLY_INVERTED:=12, 	(* The algorithm searches for codes only in the inverted image. *)
	TCVN_CSS_FIRST_INVERTED:=14, 	(* The algorithm first searches for codes in the inverted and then in the non-inverted image. *)
	TCVN_CSS_ONLY_NOT_FLIPPED:=64, 	(* The algorithm searches for codes only in the non-mirrored image. *)
	TCVN_CSS_FIRST_NOT_FLIPPED:=80, 	(* The algorithm first searches for codes in the non-mirrored and then in the mirrored image. *)
	TCVN_CSS_ONLY_FLIPPED:=96, 	(* The algorithm searches for codes only in the mirrored image. *)
	TCVN_CSS_FIRST_FLIPPED:=112	(* The algorithm first searches for codes in the mirrored and then in the non-mirrored image. *)
) UDINT;
END_TYPE

// Data Types/Enumerations/ETcVnAdaptiveThresholdMethod

(* Offers methods for adaptive threshold. *)
	{attribute 'TcIecLibraryType'}
{attribute 'Namespace' := 'Tc3_Vision'}
TYPE ETcVnAdaptiveThresholdMethod : (
	TCVN_ATM_MEAN:=0, 	(* The threshold value is calculated as the mean of the nBlockSize x nBlockSize neighborhood of (x,y) minus fConstant. *)
	TCVN_ATM_GAUSSIAN:=1	(* The threshold value is the weighted sum (cross-correlation with a Gaussian window) of the nBlockSize x nBlockSize neighborhood of (x,y) minus fConstant. *)
) DINT;
END_TYPE

// Data Types/Enumerations/ETcVnBarcodeSearchDirection

(* Offers search directions for linear barcodes. *)
	{attribute 'TcIecLibraryType'}
{attribute 'Namespace' := 'Tc3_Vision'}
TYPE ETcVnBarcodeSearchDirection : (
	TCVN_BSD_ANY:=0, 	(* The algorithm searches for codes in any supported directions. *)
	TCVN_BSD_HORIZONTAL:=1, 	(* The algorithm searches for codes in horizontal direction. *)
	TCVN_BSD_VERTICAL:=2	(* The algorithm searches for codes in vertical direction. *)
) UDINT;
END_TYPE

// Data Types/Enumerations/ETcVnBarcodeType

(* Offers linear barcode types to search for. *)
	{attribute 'TcIecLibraryType'}
{attribute 'Namespace' := 'Tc3_Vision'}
TYPE ETcVnBarcodeType : (
	TCVN_BT_CODABAR:=4, 	(* The algorithm searches for Codabar codes. *)
	TCVN_BT_CODE39:=8, 	(* The algorithm searches for Code-39 codes. *)
	TCVN_BT_CODE93:=16, 	(* The algorithm searches for Code-93 codes. *)
	TCVN_BT_CODE128:=32, 	(* The algorithm searches for Code-128 codes. *)
	TCVN_BT_EAN8:=128, 	(* The algorithm searches for EAN-8 codes. *)
	TCVN_BT_EAN13:=256, 	(* The algorithm searches for EAN-13 codes. *)
	TCVN_BT_ITF:=512, 	(* The algorithm searches for ITF codes. *)
	TCVN_BT_UPCA:=32768, 	(* The algorithm searches for UPC-A codes. *)
	TCVN_BT_UPCE:=65536, 	(* The algorithm searches for UPC-E codes. *)
	TCVN_BT_ANY:=99260, 	(* The algorithm searches for any supported linear barcode. If the type of the code is known, it is recommended to select the specific type directly. *)
	TCVN_BT_CODE39EXTENDED:=262144	(* The algorithm searches for Code-93-Extended codes. *)
) UDINT;
END_TYPE

// Data Types/Enumerations/ETcVnBlobCombination

(* Offers multiple blob contours to choose from, which should be returned in a multi-threshold scenario (used in TcVnParamsBlobDetection, which in return is used in F_VN_DetectBlobs). *)
	{attribute 'TcIecLibraryType'}
{attribute 'Namespace' := 'Tc3_Vision'}
TYPE ETcVnBlobCombination : (
	TCVN_BC_SMALLEST:=0, 	(* Returns the smallest blob contour. *)
	TCVN_BC_LARGEST:=1, 	(* Returns the largest blob contour. *)
	TCVN_BC_MIN_THRESHOLD:=2, 	(* Returns the blob contour for the minimum threshold. *)
	TCVN_BC_MAX_THRESHOLD:=3, 	(* Returns the blob contour for the maximum threshold. *)
	TCVN_BC_MEDIAN_THRESHOLD:=4	(* Returns the blob contour for the median threshold. *)
) DINT;
END_TYPE

// Data Types/Enumerations/ETcVnBoostClassifierType

(* Offers different types of Boost classifiers. *)
	{attribute 'TcIecLibraryType'}
{attribute 'Namespace' := 'Tc3_Vision'}
TYPE ETcVnBoostClassifierType : (
	TCVN_BCT_DISCRETE:=0, 	(* Discrete AdaBoost *)
	TCVN_BCT_REAL:=1, 	(* Real AdaBoost *)
	TCVN_BCT_LOGIT:=2, 	(* LogitBoost *)
	TCVN_BCT_GENTLE:=3	(* Gentle AdaBoost *)
) DINT;
END_TYPE

// Data Types/Enumerations/ETcVnBorderInterpolationMethod

(* Offers methods to extrapolate values of non-existing pixels. On the one hand, this is used for filtering functions to enable filtering at the image borders (where the filter mask reaches over the border). On the other hand, this is used to extrapolate the undefined pixels after a geometric image transformation. *)
	{attribute 'TcIecLibraryType'}
{attribute 'Namespace' := 'Tc3_Vision'}
{warning disable C0125}
TYPE ETcVnBorderInterpolationMethod : (
	TCVN_BIM_CONSTANT:=0, 	(* iiiiiii | abcdefgh | iiiiiii  (with some specified i) *)
	TCVN_BIM_REPLICATE:=1, 	(* aaaaaaa | abcdefgh | hhhhhhh *)
	TCVN_BIM_REFLECT:=2, 	(* gfedcba | abcdefgh | hgfedcb *)
	TCVN_BIM_WRAP:=3, 	(* bcdefgh | abcdefgh | abcdefg *)
	TCVN_BIM_REFLECT_101:=4, 	(* hgfedcb | abcdefgh | gfedcba *)
	TCVN_BIM_DEFAULT:=4, 	(* Choose this if you don't know which method to select (same as REFLECT_101). *)
	TCVN_BIM_TRANSPARENT:=5, 	(* Corresponding pixels in the destination image will not be modified. Only available for geometric image transformations. *)
	TCVN_BIM_ISOLATED_CONSTANT:=16, 	(* Similar to CONSTANT, but ROIs are handled as isolated, which means surrounding image pixels outside the ROI are ignored. *)
	TCVN_BIM_ISOLATED_REPLICATE:=17, 	(* Similar to REPLICATE, but ROIs are handled as isolated, which means surrounding image pixels outside the ROI are ignored. *)
	TCVN_BIM_ISOLATED_REFLECT:=18, 	(* Similar to REFLECT, but ROIs are handled as isolated, which means surrounding image pixels outside the ROI are ignored. *)
	TCVN_BIM_ISOLATED_WRAP:=19, 	(* Similar to WRAP, but ROIs are handled as isolated, which means surrounding image pixels outside the ROI are ignored. *)
	TCVN_BIM_ISOLATED_REFLECT_101:=20	(* Similar to REFLECT_101, but ROIs are handled as isolated, which means surrounding image pixels outside the ROI are ignored. *)
) DINT;
END_TYPE

// Data Types/Enumerations/ETcVnCalibrationPattern

(* Offers common calibration pattern types. *)
	{attribute 'TcIecLibraryType'}
{attribute 'Namespace' := 'Tc3_Vision'}
TYPE ETcVnCalibrationPattern : (
	TCVN_CP_CIRCLES_SYM:=0, 	(* Symmetric circle pattern *)
	TCVN_CP_CIRCLES_ASYM:=1, 	(* Asymmetric circle pattern, i.e. every 2nd row is indented, starting unindented *)
	TCVN_CP_CIRCLES_ASYM_INDENT:=2	(* Asymmetric circle pattern, i.e. every 2nd row is indented, starting indented *)
) DINT;
END_TYPE

// Data Types/Enumerations/ETcVnCalibrationPatternOrigin

(* Offers calibration pattern origins. *)
	{attribute 'TcIecLibraryType'}
{attribute 'Namespace' := 'Tc3_Vision'}
TYPE ETcVnCalibrationPatternOrigin : (
	TCVN_CPO_TOPLEFT:=0, 	(* Origin is at top left *)
	TCVN_CPO_TOPCENTER:=1, 	(* Origin is at top center *)
	TCVN_CPO_TOPRIGHT:=2, 	(* Origin is at top right *)
	TCVN_CPO_CENTERLEFT:=3, 	(* Origin is at center left *)
	TCVN_CPO_CENTER:=4, 	(* Origin is at center *)
	TCVN_CPO_CENTERRIGHT:=5, 	(* Origin is at center right *)
	TCVN_CPO_BOTTOMLEFT:=6, 	(* Origin is at bottom left *)
	TCVN_CPO_BOTTOMCENTER:=7, 	(* Origin is at bottom center *)
	TCVN_CPO_BOTTOMRIGHT:=8	(* Origin is at bottom right *)
) DINT;
END_TYPE

// Data Types/Enumerations/ETcVnCameraState

(* Specifies the state of a camera controller, which controls an attached camera. *)
	{attribute 'TcIecLibraryType'}
{attribute 'Namespace' := 'Tc3_Vision'}
TYPE ETcVnCameraState : (
	TCVN_CS_ERROR:=-1, 	(* The camera controller is in an error state (e.g. the connection to the camera was lost). *)
	TCVN_CS_INITIAL:=0, 	(* The camera controller is in the initial state and ready to establish the connection to the camera. *)
	TCVN_CS_INITIALIZING:=1, 	(* The camera controller is initializing the camera. *)
	TCVN_CS_INITIALIZED:=2, 	(* The camera controller has initialized the camera. *)
	TCVN_CS_OPENING:=3, 	(* The camera controller is establishing the connection to the camera. *)
	TCVN_CS_OPENED:=4, 	(* The connection to the camera has been established and the camera controller is ready to start the image acquisition. *)
	TCVN_CS_STARTACQUISITION:=5, 	(* The camera controller is starting the image acquisition. *)
	TCVN_CS_ACQUIRING:=6, 	(* The camera is sending images (either streaming or manually triggered, depending on the configuration). *)
	TCVN_CS_STOPACQUISITION:=7, 	(* The camera controller is stopping the image acquisition. *)
	TCVN_CS_RESETTINGFEATURES:=8, 	(* The camera controller is resetting the features on the camera. *)
	TCVN_CS_TRIGGERING:=9, 	(* The camera controller is processing a softwaretrigger. *)
	TCVN_CS_CLOSING:=10	(* The camera controller is closing the connection to the camera. *)
) DINT;
END_TYPE

// Data Types/Enumerations/ETcVnClusteringAlgorithm

(* Offers clustering algorithms *)
	{attribute 'TcIecLibraryType'}
{attribute 'Namespace' := 'Tc3_Vision'}
TYPE ETcVnClusteringAlgorithm : (
	TCVN_CA_KMEANSPP:=0, 	(* KMeans++ (fixed number of clusters) *)
	TCVN_CA_LBG:=1	(* LBG variant (dynamic number of clusters) *)
) DINT;
END_TYPE

// Data Types/Enumerations/ETcVnColorMap

(* Offers color maps (similar to GNU Octave/MATLAB types). *)
	{attribute 'TcIecLibraryType'}
{attribute 'Namespace' := 'Tc3_Vision'}
TYPE ETcVnColorMap : (
	TCVN_CM_AUTUMN:=0, 	(* Red - orange - yellow *)
	TCVN_CM_BONE:=1, 	(* Black - blueish gray - white *)
	TCVN_CM_JET:=2, 	(* Dark blue - green - dark red *)
	TCVN_CM_WINTER:=3, 	(* Blue - green *)
	TCVN_CM_RAINBOW:=4, 	(* Red - green - purple *)
	TCVN_CM_OCEAN:=5, 	(* Black - blue - white *)
	TCVN_CM_SUMMER:=6, 	(* Green - yellow *)
	TCVN_CM_SPRING:=7, 	(* Pink - yellow *)
	TCVN_CM_COOL:=8, 	(* Cyan - magenta *)
	TCVN_CM_HSV:=9, 	(* Red - green - blue - red *)
	TCVN_CM_PINK:=10, 	(* Black - pink - light yellow - white *)
	TCVN_CM_HOT:=11, 	(* Black - red - yellow - white *)
	TCVN_CM_PARULA:=12, 	(* Blue - yellow *)
	TCVN_CM_MAGMA:=13, 	(* Black - magenta - light yellow *)
	TCVN_CM_INFERNO:=14, 	(* Black - magenta - yellow *)
	TCVN_CM_PLASMA:=15, 	(* Blue - magenta - yellow *)
	TCVN_CM_VIRIDIS:=16, 	(* Purple - yellow *)
	TCVN_CM_CIVIDIS:=17, 	(* Blue - gray - yellow *)
	TCVN_CM_TWILIGHT:=18, 	(* White - light blue - dark purple - light red - white *)
	TCVN_CM_TWILIGHT_SHIFTED:=19, 	(* Dark purple - light blue - white - light red - dark purple *)
	TCVN_CM_TURBO:=20	(* Dark blue - light green - dark red *)
) DINT;
END_TYPE

// Data Types/Enumerations/ETcVnColorMapSize

(* Offers color map sizes. *)
	{attribute 'TcIecLibraryType'}
{attribute 'Namespace' := 'Tc3_Vision'}
TYPE ETcVnColorMapSize : (
	TCVN_CMS_256:=256, 	(* 256 colors, used for 8 bit images (TCVN_ET_USINT) *)
	TCVN_CMS_65536:=65536	(* 65536 colors, used for 16 bit images (TCVN_ET_UINT) *)
) UDINT;
END_TYPE

// Data Types/Enumerations/ETcVnColorSpaceTransform

(* Offers color space transformations. *)
	{attribute 'TcIecLibraryType'}
{attribute 'Namespace' := 'Tc3_Vision'}
{warning disable C0125}
TYPE ETcVnColorSpaceTransform : (
	TCVN_CST_BGR_TO_BGRA:=0, 	(* Transform the color space from BGR to BGRA. *)
	TCVN_CST_RGB_TO_RGBA:=0, 	(* Transform the color space from RGB to RGBA. *)
	TCVN_CST_BGRA_TO_BGR:=1, 	(* Transform the color space from BGRA to BGR. *)
	TCVN_CST_RGBA_TO_RGB:=1, 	(* Transform the color space from RGBA to RGB. *)
	TCVN_CST_BGR_TO_RGBA:=2, 	(* Transform the color space from BGR to RGBA. *)
	TCVN_CST_RGB_TO_BGRA:=2, 	(* Transform the color space from RGB to BGRA. *)
	TCVN_CST_BGRA_TO_RGB:=3, 	(* Transform the color space from BGRA to RGB. *)
	TCVN_CST_RGBA_TO_BGR:=3, 	(* Transform the color space from RGBA to BGR. *)
	TCVN_CST_BGR_TO_RGB:=4, 	(* Transform the color space from BGR to RGB. *)
	TCVN_CST_RGB_TO_BGR:=4, 	(* Transform the color space from RGB to BGR. *)
	TCVN_CST_BGRA_TO_RGBA:=5, 	(* Transform the color space from BGRA to RGBA. *)
	TCVN_CST_RGBA_TO_BGRA:=5, 	(* Transform the color space from RGBA to BGRA. *)
	TCVN_CST_BGR_TO_GRAY:=6, 	(* Transform the color space from BGR to Gray. *)
	TCVN_CST_RGB_TO_GRAY:=7, 	(* Transform the color space from RGB to Gray. *)
	TCVN_CST_GRAY_TO_BGR:=8, 	(* Transform the color space from Gray to BGR. *)
	TCVN_CST_GRAY_TO_RGB:=8, 	(* Transform the color space from Gray to RGB. *)
	TCVN_CST_GRAY_TO_BGRA:=9, 	(* Transform the color space from Gray to BGRA. *)
	TCVN_CST_GRAY_TO_RGBA:=9, 	(* Transform the color space from Gray to RGBA. *)
	TCVN_CST_BGRA_TO_GRAY:=10, 	(* Transform the color space from BGRA to Gray. *)
	TCVN_CST_RGBA_TO_GRAY:=11, 	(* Transform the color space from RGBA to Gray. *)
	TCVN_CST_RGB_TO_BGR_565:=12, 	(* Transform the color space from RGB(24 bit 888) to BGR(16 bit 565). *)
	TCVN_CST_BGR_TO_BGR_565:=13, 	(* Transform the color space from BGR(24 bit 888) to BGR(16 bit 565). *)
	TCVN_CST_BGR_565_TO_RGB:=14, 	(* Transform the color space from BGR(16 bit 565) to RGB(24 bit 888). *)
	TCVN_CST_BGR_565_TO_BGR:=15, 	(* Transform the color space from BGR(16 bit 565) to BGR(24 bit 888). *)
	TCVN_CST_RGBA_TO_BGR_565:=16, 	(* Transform the color space from RGBA(32 bit 8888) to BGR(16 bit 565). *)
	TCVN_CST_BGRA_TO_BGR_565:=17, 	(* Transform the color space from BGRA(32 bit 8888) to BGR(16 bit 565). *)
	TCVN_CST_BGR_565_TO_RGBA:=18, 	(* Transform the color space from BGR(16 bit 565) to RGBA(32 bit 8888). *)
	TCVN_CST_BGR_565_TO_BGRA:=19, 	(* Transform the color space from BGR(16 bit 565) to BGRA(32 bit 8888). *)
	TCVN_CST_GRAY_TO_BGR_565:=20, 	(* Transform the color space from Gray to BGR(16 bit 565). *)
	TCVN_CST_BGR_565_TO_GRAY:=21, 	(* Transform the color space from BGR(16 bit 565) to Gray. *)
	TCVN_CST_RGB_TO_BGR_555:=22, 	(* Transform the color space from RGB(24 bit 888) to BGR(16 bit 555). *)
	TCVN_CST_BGR_TO_BGR_555:=23, 	(* Transform the color space from BGR(24 bit 888) to BGR(16 bit 555). *)
	TCVN_CST_BGR_555_TO_RGB:=24, 	(* Transform the color space from BGR(16 bit 555) to RGB(24 bit 888). *)
	TCVN_CST_BGR_555_TO_BGR:=25, 	(* Transform the color space from BGR(16 bit 555) to BGR(24 bit 888). *)
	TCVN_CST_RGBA_TO_BGR_555:=26, 	(* Transform the color space from RGBA(32 bit 8888) to BGR(16 bit 555). *)
	TCVN_CST_BGRA_TO_BGR_555:=27, 	(* Transform the color space from BGRA(32 bit 8888) to BGR(16 bit 555). *)
	TCVN_CST_BGR_555_TO_RGBA:=28, 	(* Transform the color space from BGR(16 bit 555) to RGBA(32 bit 8888). *)
	TCVN_CST_BGR_555_TO_BGRA:=29, 	(* Transform the color space from BGR(16 bit 555) to BGRA(32 bit 8888). *)
	TCVN_CST_GRAY_TO_BGR_555:=30, 	(* Transform the color space from Gray to BGR(16 bit 555). *)
	TCVN_CST_BGR_555_TO_GRAY:=31, 	(* Transform the color space from BGR(16 bit 555) to Gray. *)
	TCVN_CST_BGR_TO_XYZ:=32, 	(* Transform the color space from BGR to CIE XYZ (scaled to the full value range of the image). *)
	TCVN_CST_RGB_TO_XYZ:=33, 	(* Transform the color space from RGB to CIE XYZ (scaled to the full value range of the image). *)
	TCVN_CST_XYZ_TO_BGR:=34, 	(* Transform the color space from CIE XYZ (scaled to the full value range of the image) to BGR. *)
	TCVN_CST_XYZ_TO_RGB:=35, 	(* Transform the color space from CIE XYZ (scaled to the full value range of the image) to RGB. *)
	TCVN_CST_BGR_TO_YCRCB:=36, 	(* Transform the color space from BGR to YCrCb (scaled to the full value range of the image). *)
	TCVN_CST_RGB_TO_YCRCB:=37, 	(* Transform the color space from RGB to YCrCb (scaled to the full value range of the image). *)
	TCVN_CST_YCRCB_TO_BGR:=38, 	(* Transform the color space from YCrCb (scaled to the full value range of the image) to BGR. *)
	TCVN_CST_YCRCB_TO_RGB:=39, 	(* Transform the color space from YCrCb (scaled to the full value range of the image) to RGB. *)
	TCVN_CST_BGR_TO_HSV:=40, 	(* Transform the color space from BGR to HSV (for images of type USINT, H is scaled to a range from 0 to 180 and S,V from 0 to 255). *)
	TCVN_CST_RGB_TO_HSV:=41, 	(* Transform the color space from RGB to HSV (for images of type USINT, H is scaled to a range from 0 to 180 and S,V from 0 to 255). *)
	TCVN_CST_BGR_TO_LAB:=44, 	(* Transform the color space from BGR to CIE L*a*b* (for images of type USINT, all channels are scaled to a range from 0 to 255). *)
	TCVN_CST_RGB_TO_LAB:=45, 	(* Transform the color space from RGB to CIE L*a*b* (for images of type USINT, all channels are scaled to a range from 0 to 255). *)
	TCVN_CST_BAYER_RG_TO_BGR:=46, 	(* Transform the color space from BayerRG to BGR. *)
	TCVN_CST_BAYER_BG_TO_RGB:=46, 	(* Transform the color space from BayerBG to RGB. *)
	TCVN_CST_BAYER_GR_TO_BGR:=47, 	(* Transform the color space from BayerGR to BGR. *)
	TCVN_CST_BAYER_GB_TO_RGB:=47, 	(* Transform the color space from BayerGB to RGB. *)
	TCVN_CST_BAYER_BG_TO_BGR:=48, 	(* Transform the color space from BayerBG to BGR. *)
	TCVN_CST_BAYER_RG_TO_RGB:=48, 	(* Transform the color space from BayerRG to RGB. *)
	TCVN_CST_BAYER_GB_TO_BGR:=49, 	(* Transform the color space from BayerGB to BGR. *)
	TCVN_CST_BAYER_GR_TO_RGB:=49, 	(* Transform the color space from BayerGR to RGB. *)
	TCVN_CST_BGR_TO_LUV:=50, 	(* Transform the color space from BGR to CIE L*u*v* (for images of type USINT, all channels are scaled to a range from 0 to 255). *)
	TCVN_CST_RGB_TO_LUV:=51, 	(* Transform the color space from RGB to CIE L*u*v* (for images of type USINT, all channels are scaled to a range from 0 to 255). *)
	TCVN_CST_BGR_TO_HLS:=52, 	(* Transform the color space from BGR to HLS (for images of type USINT, H is scaled to a range from 0 to 180 and L,S from 0 to 255). *)
	TCVN_CST_RGB_TO_HLS:=53, 	(* Transform the color space from RGB to HLS (for images of type USINT, H is scaled to a range from 0 to 180 and L,S from 0 to 255). *)
	TCVN_CST_HSV_TO_BGR:=54, 	(* Transform the color space from HSV (for images of type USINT, H is scaled to a range from 0 to 180 and S,V from 0 to 255) to BGR. *)
	TCVN_CST_HSV_TO_RGB:=55, 	(* Transform the color space from HSV (for images of type USINT, H is scaled to a range from 0 to 180 and S,V from 0 to 255) to RGB. *)
	TCVN_CST_LAB_TO_BGR:=56, 	(* Transform the color space from CIE L*a*b* (for images of type USINT, all channels are scaled to a range from 0 to 255) to BGR. *)
	TCVN_CST_LAB_TO_RGB:=57, 	(* Transform the color space from CIE L*a*b* (for images of type USINT, all channels are scaled to a range from 0 to 255) to RGB. *)
	TCVN_CST_LUV_TO_BGR:=58, 	(* Transform the color space from CIE L*u*v* (for images of type USINT, all channels are scaled to a range from 0 to 255) to BGR. *)
	TCVN_CST_LUV_TO_RGB:=59, 	(* Transform the color space from CIE L*u*v* (for images of type USINT, all channels are scaled to a range from 0 to 255) to RGB. *)
	TCVN_CST_HLS_TO_BGR:=60, 	(* Transform the color space from HLS (for images of type USINT, H is scaled to a range from 0 to 180 and L,S from 0 to 255) to BGR. *)
	TCVN_CST_HLS_TO_RGB:=61, 	(* Transform the color space from HLS (for images of type USINT, H is scaled to a range from 0 to 180 and L,S from 0 to 255) to RGB. *)
	TCVN_CST_BAYER_RG_TO_BGR_VNG:=62, 	(* Transform the color space from BayerRG to BGR, using Variable Number of Gradients. *)
	TCVN_CST_BAYER_GR_TO_BGR_VNG:=63, 	(* Transform the color space from BayerGR to BGR, using Variable Number of Gradients. *)
	TCVN_CST_BAYER_BG_TO_BGR_VNG:=64, 	(* Transform the color space from BayerBG to BGR, using Variable Number of Gradients. *)
	TCVN_CST_BAYER_GB_TO_BGR_VNG:=65, 	(* Transform the color space from BayerGB to BGR, using Variable Number of Gradients. *)
	TCVN_CST_BAYER_RG_TO_RGB_VNG:=64, 	(* Transform the color space from BayerRG to RGB, using Variable Number of Gradients. *)
	TCVN_CST_BAYER_GR_TO_RGB_VNG:=65, 	(* Transform the color space from BayerGR to RGB, using Variable Number of Gradients. *)
	TCVN_CST_BAYER_BG_TO_RGB_VNG:=62, 	(* Transform the color space from BayerBG to RGB, using Variable Number of Gradients. *)
	TCVN_CST_BAYER_GB_TO_RGB_VNG:=63, 	(* Transform the color space from BayerGB to RGB, using Variable Number of Gradients. *)
	TCVN_CST_BGR_TO_HSV_FULL:=66, 	(* Transform the color space from BGR to HSV (for images of type USINT, all channels are scaled to a range from 0 to 255). *)
	TCVN_CST_RGB_TO_HSV_FULL:=67, 	(* Transform the color space from RGB to HSV (for images of type USINT, all channels are scaled to a range from 0 to 255). *)
	TCVN_CST_BGR_TO_HLS_FULL:=68, 	(* Transform the color space from BGR to HLS (for images of type USINT, all channels are scaled to a range from 0 to 255). *)
	TCVN_CST_RGB_TO_HLS_FULL:=69, 	(* Transform the color space from RGB to HLS (for images of type USINT, all channels are scaled to a range from 0 to 255). *)
	TCVN_CST_HSV_TO_BGR_FULL:=70, 	(* Transform the color space from HSV (for images of type USINT, all channels are scaled to a range from 0 to 255) to BGR. *)
	TCVN_CST_HSV_TO_RGB_FULL:=71, 	(* Transform the color space from HSV (for images of type USINT, all channels are scaled to a range from 0 to 255) to RGB. *)
	TCVN_CST_HLS_TO_BGR_FULL:=72, 	(* Transform the color space from HLS (for images of type USINT, all channels are scaled to a range from 0 to 255) to BGR. *)
	TCVN_CST_HLS_TO_RGB_FULL:=73, 	(* Transform the color space from HLS (for images of type USINT, all channels are scaled to a range from 0 to 255) to RGB. *)
	TCVN_CST_LBGR_TO_LAB:=74, 	(* Transform the color space from LBGR to CIE L*a*b* (for images of type USINT, all channels are scaled to a range from 0 to 255). *)
	TCVN_CST_LRGB_TO_LAB:=75, 	(* Transform the color space from LRGB to CIE L*a*b* (for images of type USINT, all channels are scaled to a range from 0 to 255). *)
	TCVN_CST_LBGR_TO_LUV:=76, 	(* Transform the color space from LBGR to CIE L*u*v* (for images of type USINT, all channels are scaled to a range from 0 to 255). *)
	TCVN_CST_LRGB_TO_LUV:=77, 	(* Transform the color space from LRGB to CIE L*u*v* (for images of type USINT, all channels are scaled to a range from 0 to 255). *)
	TCVN_CST_LAB_TO_LBGR:=78, 	(* Transform the color space from CIE L*a*b* (for images of type USINT, all channels are scaled to a range from 0 to 255) to LBGR. *)
	TCVN_CST_LAB_TO_LRGB:=79, 	(* Transform the color space from CIE L*a*b* (for images of type USINT, all channels are scaled to a range from 0 to 255) to LRGB. *)
	TCVN_CST_LUV_TO_LBGR:=80, 	(* Transform the color space from CIE L*u*v* (for images of type USINT, all channels are scaled to a range from 0 to 255) to LBGR. *)
	TCVN_CST_LUV_TO_LRGB:=81, 	(* Transform the color space from CIE L*u*v* (for images of type USINT, all channels are scaled to a range from 0 to 255) to LRGB. *)
	TCVN_CST_BGR_TO_YUV:=82, 	(* Transform the color space from BGR to YUV (scaled to the full value range of the image). *)
	TCVN_CST_RGB_TO_YUV:=83, 	(* Transform the color space from RGB to YUV (scaled to the full value range of the image). *)
	TCVN_CST_YUV_TO_BGR:=84, 	(* Transform the color space from YUV (scaled to the full value range of the image) to BGR. *)
	TCVN_CST_YUV_TO_RGB:=85, 	(* Transform the color space from YUV (scaled to the full value range of the image) to RGB. *)
	TCVN_CST_BAYER_RG_TO_GRAY:=86, 	(* Transform the color space from BayerRG to Gray. *)
	TCVN_CST_BAYER_GR_TO_GRAY:=87, 	(* Transform the color space from BayerGR to Gray. *)
	TCVN_CST_BAYER_BG_TO_GRAY:=88, 	(* Transform the color space from BayerBG to Gray. *)
	TCVN_CST_BAYER_GB_TO_GRAY:=89, 	(* Transform the color space from BayerGB to Gray. *)
	TCVN_CST_YUV_420_NV12_TO_RGB:=90, 	(* Transform the color space from YUV420 NV12 to RGB. *)
	TCVN_CST_YUV_420_NV12_TO_BGR:=91, 	(* Transform the color space from YUV420 NV12 to BGR. *)
	TCVN_CST_YUV_420_NV21_TO_RGB:=92, 	(* Transform the color space from YUV420 NV21 (SP) to RGB. *)
	TCVN_CST_YUV_420_NV21_TO_BGR:=93, 	(* Transform the color space from YUV420 NV21 (SP) to BGR. *)
	TCVN_CST_YUV_420_SP_TO_RGB:=92, 	(* Transform the color space from YUV420 NV21 (SP) to RGB. *)
	TCVN_CST_YUV_420_SP_TO_BGR:=93, 	(* Transform the color space from YUV420 NV21 (SP) to BGR. *)
	TCVN_CST_YUV_420_NV12_TO_RGBA:=94, 	(* Transform the color space from YUV420 NV12 to RGBA. *)
	TCVN_CST_YUV_420_NV12_TO_BGRA:=95, 	(* Transform the color space from YUV420 NV12 to BGRA. *)
	TCVN_CST_YUV_420_NV21_TO_RGBA:=96, 	(* Transform the color space from YUV420 NV21 (SP) to RGBA. *)
	TCVN_CST_YUV_420_NV21_TO_BGRA:=97, 	(* Transform the color space from YUV420 NV21 (SP) to BGRA. *)
	TCVN_CST_YUV_420_SP_TO_RGBA:=96, 	(* Transform the color space from YUV420 NV21 (SP) to RGBA. *)
	TCVN_CST_YUV_420_SP_TO_BGRA:=97, 	(* Transform the color space from YUV420 NV21 (SP) to BGRA. *)
	TCVN_CST_YUV_420_YV12_TO_RGB:=98, 	(* Transform the color space from YUV420 YV12 (P) to RGB. *)
	TCVN_CST_YUV_420_YV12_TO_BGR:=99, 	(* Transform the color space from YUV420 YV12 (P) to BGR. *)
	TCVN_CST_YUV_420_IYUV_TO_RGB:=100, 	(* Transform the color space from YUV420 IYUV (I420) to RGB. *)
	TCVN_CST_YUV_420_IYUV_TO_BGR:=101, 	(* Transform the color space from YUV420 IYUV (I420) to BGR. *)
	TCVN_CST_YUV_420_I420_TO_RGB:=100, 	(* Transform the color space from YUV420 IYUV (I420) to RGB. *)
	TCVN_CST_YUV_420_I420_TO_BGR:=101, 	(* Transform the color space from YUV420 IYUV (I420) to BGR. *)
	TCVN_CST_YUV_420_P_TO_RGB:=98, 	(* Transform the color space from YUV420 YV12 (P) to RGB. *)
	TCVN_CST_YUV_420_P_TO_BGR:=99, 	(* Transform the color space from YUV420 YV12 (P) to BGR. *)
	TCVN_CST_YUV_420_YV12_TO_RGBA:=102, 	(* Transform the color space from YUV420 YV12 (P) to RGBA. *)
	TCVN_CST_YUV_420_YV12_TO_BGRA:=103, 	(* Transform the color space from YUV420 YV12 (P) to BGRA. *)
	TCVN_CST_YUV_420_IYUV_TO_RGBA:=104, 	(* Transform the color space from YUV420 IYUV (I420) to RGBA. *)
	TCVN_CST_YUV_420_IYUV_TO_BGRA:=105, 	(* Transform the color space from YUV420 IYUV (I420) to BGRA. *)
	TCVN_CST_YUV_420_I420_TO_RGBA:=104, 	(* Transform the color space from YUV420 IYUV (I420) to RGBA. *)
	TCVN_CST_YUV_420_I420_TO_BGRA:=105, 	(* Transform the color space from YUV420 IYUV (I420) to BGRA. *)
	TCVN_CST_YUV_420_P_TO_RGBA:=102, 	(* Transform the color space from YUV420 YV12 (P) to RGBA. *)
	TCVN_CST_YUV_420_P_TO_BGRA:=103, 	(* Transform the color space from YUV420 YV12 (P) to BGRA. *)
	TCVN_CST_YUV_420_TO_GRAY:=106, 	(* Transform the color space from YUV420 to Gray. *)
	TCVN_CST_YUV_420_NV21_TO_GRAY:=106, 	(* Transform the color space from YUV420 to Gray. *)
	TCVN_CST_YUV_420_NV12_TO_GRAY:=106, 	(* Transform the color space from YUV420 to Gray. *)
	TCVN_CST_YUV_420_YV12_TO_GRAY:=106, 	(* Transform the color space from YUV420 to Gray. *)
	TCVN_CST_YUV_420_IYUV_TO_GRAY:=106, 	(* Transform the color space from YUV420 to Gray. *)
	TCVN_CST_YUV_420_I420_TO_GRAY:=106, 	(* Transform the color space from YUV420 to Gray. *)
	TCVN_CST_YUV_420_SP_TO_GRAY:=106, 	(* Transform the color space from YUV420 to Gray. *)
	TCVN_CST_YUV_420_P_TO_GRAY:=106, 	(* Transform the color space from YUV420 to Gray. *)
	TCVN_CST_YUV_422_UYVY_TO_RGB:=107, 	(* Transform the color space from YUV422 UYVY (Y422, UYNV) to RGB. *)
	TCVN_CST_YUV_422_UYVY_TO_BGR:=108, 	(* Transform the color space from YUV422 UYVY (Y422, UYNV) to BGR. *)
	TCVN_CST_YUV_422_Y422_TO_RGB:=107, 	(* Transform the color space from YUV422 UYVY (Y422, UYNV) to RGB. *)
	TCVN_CST_YUV_422_Y422_TO_BGR:=108, 	(* Transform the color space from YUV422 UYVY (Y422, UYNV) to BGR. *)
	TCVN_CST_YUV_422_UYNV_TO_RGB:=107, 	(* Transform the color space from YUV422 UYVY (Y422, UYNV) to RGB. *)
	TCVN_CST_YUV_422_UYNV_TO_BGR:=108, 	(* Transform the color space from YUV422 UYVY (Y422, UYNV) to BGR. *)
	TCVN_CST_YUV_422_UYVY_TO_RGBA:=111, 	(* Transform the color space from YUV422 UYVY (Y422, UYNV) to RGBA. *)
	TCVN_CST_YUV_422_UYVY_TO_BGRA:=112, 	(* Transform the color space from YUV422 UYVY (Y422, UYNV) to BGRA. *)
	TCVN_CST_YUV_422_Y422_TO_RGBA:=111, 	(* Transform the color space from YUV422 UYVY (Y422, UYNV) to RGB. *)
	TCVN_CST_YUV_422_Y422_TO_BGRA:=112, 	(* Transform the color space from YUV422 UYVY (Y422, UYNV) to BGRA. *)
	TCVN_CST_YUV_422_UYNV_TO_RGBA:=111, 	(* Transform the color space from YUV422 UYVY (Y422, UYNV) to RGB. *)
	TCVN_CST_YUV_422_UYNV_TO_BGRA:=112, 	(* Transform the color space from YUV422 UYVY (Y422, UYNV) to BGRA. *)
	TCVN_CST_YUV_422_YUY2_TO_RGB:=115, 	(* Transform the color space from YUV422 YUYV (YUY2, YUNV) to RGB. *)
	TCVN_CST_YUV_422_YUY2_TO_BGR:=116, 	(* Transform the color space from YUV422 YUYV (YUY2, YUNV) to BGR. *)
	TCVN_CST_YUV_422_YVYU_TO_RGB:=117, 	(* Transform the color space from YUV422 YVYU to RGB. *)
	TCVN_CST_YUV_422_YVYU_TO_BGR:=118, 	(* Transform the color space from YUV422 YVYU to BGR. *)
	TCVN_CST_YUV_422_YUYV_TO_RGB:=115, 	(* Transform the color space from YUV422 YUYV (YUY2, YUNV) to RGB. *)
	TCVN_CST_YUV_422_YUYV_TO_BGR:=116, 	(* Transform the color space from YUV422 YUYV (YUY2, YUNV) to BGR. *)
	TCVN_CST_YUV_422_YUNV_TO_RGB:=115, 	(* Transform the color space from YUV422 YUYV (YUY2, YUNV) to RGB. *)
	TCVN_CST_YUV_422_YUNV_TO_BGR:=116, 	(* Transform the color space from YUV422 YUYV (YUY2, YUNV) to BGR. *)
	TCVN_CST_YUV_422_YUY2_TO_RGBA:=119, 	(* Transform the color space from YUV422 YUYV (YUY2, YUNV) to RGBA. *)
	TCVN_CST_YUV_422_YUY2_TO_BGRA:=120, 	(* Transform the color space from YUV422 YUYV (YUY2, YUNV) to BGRA. *)
	TCVN_CST_YUV_422_YVYU_TO_RGBA:=121, 	(* Transform the color space from YUV422 YVYU to RGBA. *)
	TCVN_CST_YUV_422_YVYU_TO_BGRA:=122, 	(* Transform the color space from YUV422 YVYU to BGRA. *)
	TCVN_CST_YUV_422_YUYV_TO_RGBA:=119, 	(* Transform the color space from YUV422 YUYV (YUY2, YUNV) to RGBA. *)
	TCVN_CST_YUV_422_YUYV_TO_BGRA:=120, 	(* Transform the color space from YUV422 YUYV (YUY2, YUNV) to BGRA. *)
	TCVN_CST_YUV_422_YUNV_TO_RGBA:=119, 	(* Transform the color space from YUV422 YUYV (YUY2, YUNV) to RGBA. *)
	TCVN_CST_YUV_422_YUNV_TO_BGRA:=120, 	(* Transform the color space from YUV422 YUYV (YUY2, YUNV) to BGRA. *)
	TCVN_CST_YUV_422_UYVY_TO_GRAY:=123, 	(* Transform the color space from YUV422 UYVY (Y422, UYNV) to Gray. *)
	TCVN_CST_YUV_422_YUY2_TO_GRAY:=124, 	(* Transform the color space from YUV422 YUYV (YUY2, YUNV) to Gray. *)
	TCVN_CST_YUV_422_Y422_TO_GRAY:=123, 	(* Transform the color space from YUV422 UYVY (Y422, UYNV) to Gray. *)
	TCVN_CST_YUV_422_UYNV_TO_GRAY:=123, 	(* Transform the color space from YUV422 UYVY (Y422, UYNV) to Gray. *)
	TCVN_CST_YUV_422_YVYU_TO_GRAY:=124, 	(* Transform the color space from YUV422 YVYU to Gray. *)
	TCVN_CST_YUV_422_YUYV_TO_GRAY:=124, 	(* Transform the color space from YUV422 YUYV (YUY2, YUNV) to Gray. *)
	TCVN_CST_YUV_422_YUNV_TO_GRAY:=124, 	(* Transform the color space from YUV422 YUYV (YUY2, YUNV) to Gray. *)
	TCVN_CST_RGBA_TO_PREMULTIPLICATED_RGBA:=125, 	(* Transform the color space from RGBA to premultiplicated RGBA. *)
	TCVN_CST_PREMULTIPLICATED_RGBA_TO_RGBA:=126, 	(* Transform the color space from premultiplicated RGBA to RGBA. *)
	TCVN_CST_RGB_TO_YUV_420_I420:=127, 	(* Transform the color space from RGB to YUV420 IYUV (I420). *)
	TCVN_CST_BGR_TO_YUV_420_I420:=128, 	(* Transform the color space from BGR to YUV420 IYUV (I420). *)
	TCVN_CST_RGB_TO_YUV_420_IYUV:=127, 	(* Transform the color space from RGB to YUV420 IYUV (I420). *)
	TCVN_CST_BGR_TO_YUV_420_IYUV:=128, 	(* Transform the color space from BGR to YUV420 IYUV (I420). *)
	TCVN_CST_RGBA_TO_YUV_420_I420:=129, 	(* Transform the color space from RGBA to YUV420 IYUV (I420). *)
	TCVN_CST_BGRA_TO_YUV_420_I420:=130, 	(* Transform the color space from BGRA to YUV420 IYUV (I420). *)
	TCVN_CST_RGBA_TO_YUV_420_IYUV:=129, 	(* Transform the color space from RGBA to YUV420 IYUV (I420). *)
	TCVN_CST_BGRA_TO_YUV_420_IYUV:=130, 	(* Transform the color space from BGRA to YUV420 IYUV (I420). *)
	TCVN_CST_RGB_TO_YUV_420_YV12:=131, 	(* Transform the color space from RGB to YUV420 YV12 (P). *)
	TCVN_CST_BGR_TO_YUV_420_YV12:=132, 	(* Transform the color space from BGR to YUV420 YV12 (P). *)
	TCVN_CST_RGBA_TO_YUV_420_YV12:=133, 	(* Transform the color space from RGBA to YUV420 YV12 (P). *)
	TCVN_CST_BGRA_TO_YUV_420_YV12:=134, 	(* Transform the color space from BGRA to YUV420 YV12 (P). *)
	TCVN_CST_BAYER_RG_TO_BGR_EA:=135, 	(* Transform the color space from BayerRG to BGR, using an Edge Aware algorithm. *)
	TCVN_CST_BAYER_GR_TO_BGR_EA:=136, 	(* Transform the color space from BayerGR to BGR, using an Edge Aware algorithm. *)
	TCVN_CST_BAYER_BG_TO_BGR_EA:=137, 	(* Transform the color space from BayerBG to BGR, using an Edge Aware algorithm. *)
	TCVN_CST_BAYER_GB_TO_BGR_EA:=138, 	(* Transform the color space from BayerGB to BGR, using an Edge Aware algorithm. *)
	TCVN_CST_BAYER_RG_TO_RGB_EA:=137, 	(* Transform the color space from BayerRG to RGB, using an Edge Aware algorithm. *)
	TCVN_CST_BAYER_GR_TO_RGB_EA:=138, 	(* Transform the color space from BayerGR to RGB, using an Edge Aware algorithm. *)
	TCVN_CST_BAYER_BG_TO_RGB_EA:=135, 	(* Transform the color space from BayerBG to RGB, using an Edge Aware algorithm. *)
	TCVN_CST_BAYER_GB_TO_RGB_EA:=136, 	(* Transform the color space from BayerGB to RGB, using an Edge Aware algorithm. *)
	TCVN_CST_BAYER_RG_TO_BGRA:=139, 	(* Transform the color space from BayerRG to BGRA. *)
	TCVN_CST_BAYER_GR_TO_BGRA:=140, 	(* Transform the color space from BayerGR to BGRA. *)
	TCVN_CST_BAYER_BG_TO_BGRA:=141, 	(* Transform the color space from BayerBG to BGRA. *)
	TCVN_CST_BAYER_GB_TO_BGRA:=142, 	(* Transform the color space from BayerGB to BGRA. *)
	TCVN_CST_BAYER_RG_TO_RGBA:=141, 	(* Transform the color space from BayerRG to RGBA. *)
	TCVN_CST_BAYER_GR_TO_RGBA:=142, 	(* Transform the color space from BayerGR to RGBA. *)
	TCVN_CST_BAYER_BG_TO_RGBA:=139, 	(* Transform the color space from BayerBG to RGBA. *)
	TCVN_CST_BAYER_GB_TO_RGBA:=140, 	(* Transform the color space from BayerGB to RGBA. *)
	TCVN_CST_MAX:=143	(* For internal use only, adapted when adding new values. *)
) DINT;
END_TYPE

// Data Types/Enumerations/ETcVnColorTrainingMethod

(* Offers color training methods. *)
	{attribute 'TcIecLibraryType'}
{attribute 'Namespace' := 'Tc3_Vision'}
TYPE ETcVnColorTrainingMethod : (
	TCVN_CTM_LAB:=0, 	(* Trains the color in CIE L*a*b* color space. *)
	TCVN_CTM_RGB:=1	(* Trains the color in RGB color space. *)
) DINT;
END_TYPE

// Data Types/Enumerations/ETcVnConnectedComponentsAlgorithm

(* Offers connected components algorithms. *)
	{attribute 'TcIecLibraryType'}
{attribute 'Namespace' := 'Tc3_Vision'}
TYPE ETcVnConnectedComponentsAlgorithm : (
	TCVN_CCA_WU:=0, 	(* SAUF algorithm *)
	TCVN_CCA_GRANA:=1	(* BBDT algorithm for 8-way connectivity, SAUF algorithm for 4-way connectivity *)
) DINT;
END_TYPE

// Data Types/Enumerations/ETcVnContainerExportFormat

(* Offers container export formats. *)
	{attribute 'TcIecLibraryType'}
{attribute 'Namespace' := 'Tc3_Vision'}
TYPE ETcVnContainerExportFormat : (
	TCVN_CEF_XML:=0, 	(* XML format with human readable data *)
	TCVN_CEF_XML_SERIALIZED:=1, 	(* XML format with serialized data *)
	TCVN_CEF_CSV:=2, 	(* CSV format (limited to two dimensional representation, so not applicable for all container types) *)
	TCVN_CEF_BINARY:=3	(* Binary serialized data (recommended for large containers) *)
) UINT;
END_TYPE

// Data Types/Enumerations/ETcVnContourApproximationMethod

(* Offers methods for contour approximation. *)
	{attribute 'TcIecLibraryType'}
{attribute 'Namespace' := 'Tc3_Vision'}
TYPE ETcVnContourApproximationMethod : (
	TCVN_CAM_NONE:=1, 	(* No approximation, every single point is stored, i.e. two subsequent points are always direct neighbors (horizontal, vertical or diagonal). *)
	TCVN_CAM_SIMPLE:=2, 	(* Lossless compression of segments that form straight lines in horizontal, vertical or diagonal direction leaving only their endpoints (For instance, an up-right rectangle is reduced to its four corner points.) *)
	TCVN_CAM_TC89_L1:=3, 	(* Compression using a Teh-Chin chain approximation algorithm (IEEE-paper C. Teh, R. Chin, On the Detection of Dominant Points on Digital Curves, 1989). *)
	TCVN_CAM_TC89_KCOS:=4	(* Compression using a Teh-Chin chain approximation algorithm (IEEE-paper C. Teh, R. Chin, On the Detection of Dominant Points on Digital Curves, 1989). *)
) DINT;
END_TYPE

// Data Types/Enumerations/ETcVnCircularityCalculationMethod

(* Offers methods to calculate contour circularity *)
	{attribute 'TcIecLibraryType'}
{attribute 'Namespace' := 'Tc3_Vision'}
TYPE ETcVnCircularityCalculationMethod : (
	TCVN_CCM_DEFAULT:=0, 	(* 4pi * area / perimeter^2 *)
	TCVN_CCM_CONVEXHULL_PERIMETER:=1, 	(* 4pi * area / (convex hull perimeter)^2 *)
	TCVN_CCM_MAX_RADIUS:=2, 	(* area / (pi * r^2), r = max distance to the contour's center of mass *)
	TCVN_CCM_ENCLOSINGCIRCLE_RADIUS:=3	(* area / (pi * r^2), r = radius of the minimum enclosing circle *)
) DINT;
END_TYPE

// Data Types/Enumerations/ETcVnContoursMatchComparisonMethod

(* Offers comparison methods for contour matching. *)
	{attribute 'TcIecLibraryType'}
{attribute 'Namespace' := 'Tc3_Vision'}
TYPE ETcVnContoursMatchComparisonMethod : (
	TCVN_CMCM_CONTOURS_MATCH_I1:=1, 	(* Contours are compared using the sum over the differences between the reciprocal individual characteristics. *)
	TCVN_CMCM_CONTOURS_MATCH_I2:=2, 	(* Contours are compared using the sum over the differences between the individual characteristics. *)
	TCVN_CMCM_CONTOURS_MATCH_I3:=3	(* Contours are compared using only the maximum difference between the individual characteristics. *)
) DINT;
END_TYPE

// Data Types/Enumerations/ETcVnContourRetrievalMode

(* Offers retrieval modes for a contour search. *)
	{attribute 'TcIecLibraryType'}
{attribute 'Namespace' := 'Tc3_Vision'}
TYPE ETcVnContourRetrievalMode : (
	TCVN_CRM_EXTERNAL:=0, 	(* Returns only external contours. *)
	TCVN_CRM_LIST:=1, 	(* Returns all found contours, not considering their hierarchy. *)
	TCVN_CRM_CONNECTED_COMPONENTS:=2, 	(* Returns all contours with a 2-level hierarchy (External contours are assigned level 0, internal contours level 1). *)
	TCVN_CRM_TREE:=3, 	(* Returns all contours and their full hierarchy. *)
	TCVN_CRM_FLOODFILL:=4	(* Returns the found contours using a floodfill algorithm (only available for DINT images). *)
) DINT;
END_TYPE

// Data Types/Enumerations/ETcVnDataLayout

(* Offers image data layouts. *)
	{attribute 'TcIecLibraryType'}
{attribute 'Namespace' := 'Tc3_Vision'}
TYPE ETcVnDataLayout : (
	TCVN_DL_DEFAULT:=16#0, 	(* Default *)
	TCVN_DL_2D_HW:=16#12, 	(* 2D data HW, multi/single channel image *)
	TCVN_DL_2D_WH:=16#21, 	(* 2D data WH, multi/single channel image *)
	TCVN_DL_3D_CHW:=16#123, 	(* 3D data CHW, single channel image *)
	TCVN_DL_3D_HWC:=16#231, 	(* 3D data HWC, single channel image *)
	TCVN_DL_4D_NCHW:=16#1234, 	(* 4D data NCHW, single channel image *)
	TCVN_DL_4D_NHWC:=16#1342	(* 4D data NHWC, single channel image *)
) ULINT;
END_TYPE

// Data Types/Enumerations/ETcVnLayerNameType

(* Offer different types of neural network model layer names *)
	{attribute 'TcIecLibraryType'}
{attribute 'Namespace' := 'Tc3_Vision'}
TYPE ETcVnLayerNameType : (
	TCVN_LNT_ALL:=0, 	(* Return the name of all layers *)
	TCVN_LNT_OUTPUTS:=1, 	(* Return the names of unconnected output layers *)
	TCVN_LNT_INPUTS:=2	(* Return the names of model inputs *)
) DINT;
END_TYPE

// Data Types/Enumerations/ETcVnDataMatrixOptions

(* Offers Data Matrix code detection options. *)
	{attribute 'TcIecLibraryType'}
{attribute 'Namespace' := 'Tc3_Vision'}
TYPE ETcVnDataMatrixOptions : (
	TCVN_DMO_DEFAULT:=0, 	(* Expects a graylevel image as input. Applies an adaptive local threshold and creates a dynamic grid based on the clock pattern. *)
	TCVN_DMO_BINARY_INPUT:=1, 	(* Expects a binary image as input (all pixels must contain 0 or 255, disables internal preprocessing) *)
	TCVN_DMO_GLOBAL_THRESHOLD:=2, 	(* Applies a global instead of an adaptive local threshold (requires uniform illumination) *)
	TCVN_DMO_BINARY_GRID:=4, 	(* Create the dynamic grid based on the binary instead of the graylevel image *)
	TCVN_DMO_STATIC_GRID:=8, 	(* Use an equally spaced static grid instead of a dynamic one *)
	TCVN_DMO_REGULAR_COLOR:=16, 	(* Only search for regular color (dark code on light background) *)
	TCVN_DMO_INVERTED_COLOR:=32	(* Only search for inverted color (light code on dark background) *)
) ULINT;
END_TYPE

// Data Types/Enumerations/ETcVnDiffusivityTypeKAZE

(* Offers diffusivity types for feature detection methods KAZE and AKAZE. *)
	{attribute 'TcIecLibraryType'}
{attribute 'Namespace' := 'Tc3_Vision'}
TYPE ETcVnDiffusivityTypeKAZE : (
	TCVN_DT1_KAZE_PM_G1:=0, 	(* Uses the Perona-Malik diffusivity filter g1. *)
	TCVN_DT1_KAZE_PM_G2:=1, 	(* Uses the Perona-Malik diffusivity filter g2. *)
	TCVN_DT1_KAZE_WEICKERT:=2, 	(* Uses the Weickert diffusivity filter. *)
	TCVN_DT1_KAZE_CHARBONNIER:=3	(* Uses the Charbonnier diffusivity filter. *)
) DINT;
END_TYPE

// Data Types/Enumerations/ETcVnDistanceTransformationLabel

(* Offers types of the label array to build. *)
	{attribute 'TcIecLibraryType'}
{attribute 'Namespace' := 'Tc3_Vision'}
TYPE ETcVnDistanceTransformationLabel : (
	TCVN_DTL_CCOMP:=0, 	(* Labels connected components (Each connected component of zeros in the source image and the pixels closest to the connected component will be assigned the same label). *)
	TCVN_DTL_PIXEL:=1	(* Labels pixels (Each zero pixel and the non-zero pixels closest to it get their own label). *)
) DINT;
END_TYPE

// Data Types/Enumerations/ETcVnDistanceTransformationMask

